    7: (* Wait 2 Seconds After Closing the Last Bin *)
        Active_Material_ID := 0;
        Active_Bin_ID := 0;
        Active_Target_Weight := 0.0;
        Status_Message := 'Settling Delay';
        Completion_Timer(IN := TRUE, PT := Post_Complete_Delay);
        IF Completion_Timer.Q THEN
            Completion_Timer(IN := FALSE);
            Step := 8; // Proceed to reset last weight
        END_IF;
        
    8: (* Reset bin_last_weight to 0 & Complete *)
        Active_Material_ID := 0;
        Active_Bin_ID := 0;
        Active_Target_Weight := 0.0;
        Status_Message := 'Sequence Completed';
        bin_last_weight := 0.0;
        Sequence_Complete := TRUE;
        
        IF NOT Start_Button THEN
            Step := 0;
            Sequence_Complete := FALSE;
            (* Reset all actual weights at completion once start is released *)
            FOR i := 1 TO 6 DO
                Actual_Weights[i] := 0.0;
            END_FOR;
        END_IF;
END_CASE;

END_FUNCTION_BLOCK

// PLC_AC500_V3/Application/old_version/Semi_Auto_Batching_V11
FUNCTION_BLOCK Semi_Auto_Batching_V11
VAR_INPUT
    Start_Button : BOOL;      // Signal to start/resume the batching sequence
    E_Stop_Active : BOOL;     // Emergency Stop (Pause/Hold signal)
    Reset : BOOL;             // Hard reset sequence back to idle state
    Semi_Auto_Bin_Material_Mapping : ARRAY[1..10] OF INT; // Material index mapping for 10 manual silos
    Semi_Auto_Bin_Cutoff_Weights : ARRAY[1..10] OF REAL; // Cutoff weight thresholds (kg)
    Semi_Auto_Bin_Tolerance : ARRAY[1..10] OF REAL; // Tolerance weight offset values (kg)
END_VAR
VAR_IN_OUT
    load_cell_value : REAL;   // Weight value read/written from load cell
END_VAR
VAR_OUTPUT
    Semi_Auto_Bin : ARRAY[1..10] OF BOOL; // Prompts/indicators for Bins 7..16
    semi_auto_bin_cutoff : ARRAY[1..10] OF BOOL; // Manual pre-cutoff indicators
    semi_auto_bin_motor : ARRAY[1..10] OF BOOL; // Main manual feeder motor outputs
    Actual_Weights : ARRAY[1..10] OF REAL; // Actual weight poured per silo
    Sequence_Complete : BOOL;  // Batch complete flag
    Active_Material_ID : INT;  // Currently active ingredient ID
    Active_Bin_ID : INT;       // Currently active physical Bin ID (7..16)
    Active_Target_Weight : REAL; // Recipe target weight of active bin (with tolerance applied)
    Error_Code : INT;          // Active error code
    Status_Message : STRING;   // Diagnostic text message
END_VAR
VAR
    Step : INT := 0;          // State machine index (0: Idle, 1..10: Bins, 11..20: Delays, 30: Settling, 40: Complete)
    bin_last_weight : REAL;   // Baseline weight snapshot before starting current bin
    actual_bin : REAL;        // Current weight added from active bin
    target_act_bin : REAL;    // Effective target weight to add from the active bin (GVL target - Tolerance)
    cutoff_trigger_weight : REAL; // Calculated target threshold weight minus cutoff and tolerance values
    Paused_By_EStop : BOOL := FALSE; // Pause status latch
    
    Mat_Idx : INT;
    i : INT;                  // General loop index
    
    (* TIMERS FOR TRANSITIONS & DELAYS *)
    Transition_Timer : TON;
    Completion_Timer : TON;
    Operator_Timer : TON;
    Step_Delay_Time : TIME := T#2S;
    Post_Complete_Delay : TIME := T#2S;
    
    (* SELF-CONTAINED SIMULATION VARIABLES *)
    Simulation_Mode : BOOL := TRUE;
    Sim_Rate : REAL := 10.0;            // Simulated pouring speed (10.0 kg/s)
    Sim_Timer : TON;
    Start_Sim_Weight : REAL;
    Discharge_Active : BOOL;
END_VAR

(* Semi-Auto Batching FB V11 with E-Stop Pause & Reset Logic *)

(* 1. HARD RESET INTERLOCK (Resets weights immediately) *)
IF Reset THEN
    FOR i := 1 TO 10 DO
        Semi_Auto_Bin[i] := FALSE;
        semi_auto_bin_cutoff[i] := FALSE;
        semi_auto_bin_motor[i] := FALSE;
        Actual_Weights[i] := 0.0;
    END_FOR;
    Sequence_Complete := FALSE;
    Active_Material_ID := 0;
    Active_Bin_ID := 0;
    Active_Target_Weight := 0.0;
    Error_Code := 0;
    Status_Message := 'Semi-Auto Reset Activated';
    Paused_By_EStop := FALSE;
    Step := 0;
    
    (* Clear simulation weights immediately *)
    load_cell_value := 0.0;
    bin_last_weight := 0.0;
    Start_Sim_Weight := 0.0;
    
    Transition_Timer(IN := FALSE);
    Completion_Timer(IN := FALSE);
    Operator_Timer(IN := FALSE);
    Sim_Timer(IN := FALSE);
    RETURN;
END_IF;

(* 2. E-STOP PAUSE / HOLD LOGIC *)
IF E_Stop_Active THEN
    Paused_By_EStop := TRUE;
END_IF;

IF Paused_By_EStop THEN
    (* Suspend all indicators and feeder outputs *)
    FOR i := 1 TO 10 DO
        Semi_Auto_Bin[i] := FALSE;
        semi_auto_bin_cutoff[i] := FALSE;
        semi_auto_bin_motor[i] := FALSE;
    END_FOR;
    
    IF E_Stop_Active THEN
        Status_Message := 'Semi-Auto Paused: Emergency Stop Active!';
    ELSE
        Status_Message := 'Semi-Auto Paused: Press Start to Resume';
        
        (* Resume sequence when Start Button is pressed *)
        IF Start_Button THEN
            Paused_By_EStop := FALSE;
        END_IF;
    END_IF;
    
    (* Freeze simulation and safety timers *)
    Sim_Timer(IN := FALSE);
    Transition_Timer(IN := FALSE);
    Completion_Timer(IN := FALSE);
    Operator_Timer(IN := FALSE);
    RETURN;
END_IF;

(* 3. SELF-CONTAINED SIMULATION WEIGHT MANAGEMENT *)
IF Simulation_Mode THEN
    (* Reset simulation to baseline *)
    IF Step = 0 AND NOT Start_Button AND NOT Sequence_Complete THEN
        load_cell_value := 0.0;
        bin_last_weight := 0.0;
        Start_Sim_Weight := 0.0;
        Sim_Timer(IN := FALSE);
    END_IF;
    
    (* Check if operator is actively pouring *)
    Discharge_Active := FALSE;
    IF Step >= 1 AND Step <= 10 THEN
        Discharge_Active := semi_auto_bin_motor[Step];
    END_IF;
    
    (* Simulate weight gain on the load cell *)
    IF Discharge_Active THEN
        Sim_Timer(IN := TRUE, PT := T#1000S);
        load_cell_value := Start_Sim_Weight + (TIME_TO_REAL(Sim_Timer.ET) / 1000.0) * Sim_Rate;
    ELSE
        Sim_Timer(IN := FALSE);
        Start_Sim_Weight := load_cell_value;
    END_IF;
END_IF;


(* 4. RECIPE SEQUENCE START *)
IF Step = 0 AND Start_Button THEN
    Step := 1;
    bin_last_weight := load_cell_value;
    Sequence_Complete := FALSE;
    Error_Code := 0;
    Status_Message := 'Semi-Auto Pour Started';
    Active_Target_Weight := 0.0;
    (* Clear actual weights on start *)
    FOR i := 1 TO 10 DO
        Actual_Weights[i] := 0.0;
        Semi_Auto_Bin[i] := FALSE;
        semi_auto_bin_cutoff[i] := FALSE;
        semi_auto_bin_motor[i] := FALSE;
    END_FOR;
END_IF;


(* 5. SEQUENCE CONTROL STATE MACHINE *)
CASE Step OF
    0:
        Active_Material_ID := 0;
        Active_Bin_ID := 0;
        Active_Target_Weight := 0.0;
        IF Error_Code = 0 THEN Status_Message := 'Semi-Auto Idle'; END_IF;
        
    1..10: (* Prompts Silos 7 to 16 *)
        Mat_Idx := Semi_Auto_Bin_Material_Mapping[Step];
        
        (* Skip this step instantly if material mapping is 0 OR target weight is 0.0 kg *)
        IF Mat_Idx = 0 OR (Mat_Idx <= 20 AND GVL.Recipe_Weights[Mat_Idx] = 0.0) THEN
            Step := Step + 1;
        ELSE
            (* Calculate effective target weight (Looked up Target - Tolerance) *)
            target_act_bin := GVL.Recipe_Weights[Mat_Idx] - Semi_Auto_Bin_Tolerance[Step];
            Active_Target_Weight := target_act_bin;
            
            (* Calculate weight added by current active bin *)
            actual_bin := load_cell_value - bin_last_weight;
            Actual_Weights[Step] := actual_bin;
            
            (* Calculate cutoff trigger threshold *)
            cutoff_trigger_weight := target_act_bin - Semi_Auto_Bin_Cutoff_Weights[Step];
            
            Active_Material_ID := Mat_Idx;
            Active_Bin_ID := Step;
            Status_Message := 'Semi-Auto Pouring Active';
            
            (* COARSE/FINE FEED TRANSITIONS WITH TOLERANCE OFFSETS *)
            IF actual_bin < cutoff_trigger_weight THEN
                (* Phase 1: Coarse Feed *)
                Semi_Auto_Bin[Step] := TRUE;
                semi_auto_bin_cutoff[Step] := FALSE;
                semi_auto_bin_motor[Step] := TRUE;
            ELSIF actual_bin < target_act_bin THEN
                (* Phase 2: Fine Feed *)
                Semi_Auto_Bin[Step] := FALSE;
                semi_auto_bin_cutoff[Step] := TRUE;
                semi_auto_bin_motor[Step] := TRUE;
            ELSE
                (* Phase 3: Completed (All OFF) *)
                Semi_Auto_Bin[Step] := FALSE;
                semi_auto_bin_cutoff[Step] := FALSE;
                semi_auto_bin_motor[Step] := FALSE;
                bin_last_weight := load_cell_value;
                Active_Target_Weight := 0.0;
                Step := 10 + Step; // Offset to separate transition states
            END_IF;
            
            (* RUNTIME CHECKS *)
            (* Check 21 & 22: Scale Limits *)
            IF load_cell_value > 500.0 THEN
                Error_Code := 21;
                Status_Message := 'Error 21: Scale Overloaded!';
                Paused_By_EStop := TRUE;
            ELSIF load_cell_value < 0.0 THEN
                Error_Code := 22;
                Status_Message := 'Error 22: Scale Underloaded/Fault!';
                Paused_By_EStop := TRUE;
            END_IF;
            
            (* Check 30: Operator Timeout *)
            Operator_Timer(IN := semi_auto_bin_motor[Step], PT := T#300S);
            IF Operator_Timer.Q THEN
                Error_Code := 30;
                Status_Message := 'Error 30: Semi-Auto Operator Timeout!';
                Paused_By_EStop := TRUE;
            END_IF;
        END_IF;

    11..19: (* Transition Delays (Between Bins) *)
        Active_Material_ID := 0;
        Active_Bin_ID := 0;
        Active_Target_Weight := 0.0;
        Status_Message := 'Transition Delay';
        Transition_Timer(IN := TRUE, PT := Step_Delay_Time);
        IF Transition_Timer.Q THEN
            Transition_Timer(IN := FALSE);
            Step := (Step - 10) + 1; // Advance to next bin
        END_IF;
        
    20: (* Transition Delay After Last Bin (Bin 10) Closes *)
        Active_Material_ID := 0;
        Active_Bin_ID := 0;
        Active_Target_Weight := 0.0;
        Status_Message := 'Settling Last Bin';
        Transition_Timer(IN := TRUE, PT := Step_Delay_Time);
        IF Transition_Timer.Q THEN
            Transition_Timer(IN := FALSE);
            Step := 30; // Go to post-discharge wait step (State 30)
        END_IF;

    30: (* Wait 2 Seconds After Closing the Last Bin *)
        Active_Material_ID := 0;
        Active_Bin_ID := 0;
        Active_Target_Weight := 0.0;
        Status_Message := 'Settling Delay';
        Completion_Timer(IN := TRUE, PT := Post_Complete_Delay);
        IF Completion_Timer.Q THEN
            Completion_Timer(IN := FALSE);
            Step := 40; // Proceed to reset last weight (State 40)
        END_IF;
        
    40: (* Reset bin_last_weight to 0 & Complete *)
        Active_Material_ID := 0;
        Active_Bin_ID := 0;
        Active_Target_Weight := 0.0;
        Status_Message := 'Sequence Completed';
        bin_last_weight := 0.0;
        Sequence_Complete := TRUE;
        
        IF NOT Start_Button THEN
            Step := 0;
            Sequence_Complete := FALSE;
            (* Reset all actual weights at completion once start is released *)
            FOR i := 1 TO 10 DO
                Actual_Weights[i] := 0.0;
            END_FOR;
        END_IF;
END_CASE;

END_FUNCTION_BLOCK

// PLC_AC500_V3/Application/old_version/Auto_Batching_V12
FUNCTION_BLOCK Auto_Batching_V12
VAR_INPUT
    Start_Button : BOOL;      // Signal to start/resume the batching sequence
    E_Stop_Active : BOOL;     // Emergency Stop (Pause/Hold signal)
    Reset : BOOL;             // Hard reset sequence back to idle state
    Auto_Bin_Material_Mapping : ARRAY[1..6] OF INT; // Material index mapping for 6 bins
    Auto_Bin_Cutoff_Weights : ARRAY[1..6] OF REAL; // Cutoff weight thresholds (kg)
    Auto_Bin_Tolerance : ARRAY[1..6] OF REAL; // Tolerance weight offset values (kg)
END_VAR
VAR_IN_OUT
    load_cell_value : REAL;   // Weight value read/written from load cell
END_VAR
VAR_OUTPUT
    Auto_Bin : ARRAY[1..6] OF BOOL; // Coarse feed valve outputs
    auto_bin_cutoff : ARRAY[1..6] OF BOOL; // Fine feed cutoff trigger indicators
    auto_bin_motor : ARRAY[1..6] OF BOOL; // Main conveyor motor outputs
    Actual_Weights : ARRAY[1..6] OF REAL; // Actual weight poured per silo
    Sequence_Complete : BOOL;  // Batch complete flag
    Active_Material_ID : INT;  // Currently active ingredient ID
    Active_Bin_ID : INT;       // Currently active physical Bin ID (1..6)
    Active_Target_Weight : REAL; // Recipe target weight of active bin (with tolerance applied)
    Error_Code : INT;          // Active error code
    Status_Message : STRING;   // Diagnostic text message
END_VAR
VAR
    Step : INT;                // State machine index
    bin_last_weight : REAL;   // Baseline weight snapshot before starting current bin
    actual_bin : REAL;        // Current weight added from active bin
    target_act_bin : REAL;    // Effective target weight to add from the active bin
    cutoff_trigger_weight : REAL; // Calculated trigger weight
    Paused_By_EStop : BOOL;    // Pause status latch
    
    Mat_Idx : INT;
    i : INT;                  // General loop index
    
    (* TIMERS FOR TRANSITIONS & DELAYS *)
    Transition_Timer : TON;
    Completion_Timer : TON;
    
    (* SELF-CONTAINED SIMULATION VARIABLES *)
    Simulation_Mode : BOOL;    // Simulation disabled
    Sim_Rate : REAL;
    Sim_Timer : TON;
    Start_Sim_Weight : REAL;
    Discharge_Active : BOOL;
END_VAR

(* Auto Batching FB V12 with E-Stop Pause & Reset Logic *)

(* 1. HARD RESET INTERLOCK (Resets weights immediately) *)
IF Reset THEN
    FOR i := 1 TO 6 DO
        Auto_Bin[i] := FALSE;
        auto_bin_cutoff[i] := FALSE;
        auto_bin_motor[i] := FALSE;
        Actual_Weights[i] := 0.0;
    END_FOR;
    Sequence_Complete := FALSE;
    Active_Material_ID := 0;
    Active_Bin_ID := 0;
    Active_Target_Weight := 0.0;
    Error_Code := 0;
    Status_Message := '';
    Paused_By_EStop := FALSE;
    Step := 0;
    
    load_cell_value := 0.0;
    bin_last_weight := 0.0;
    Start_Sim_Weight := 0.0;
    
    Transition_Timer(IN := FALSE);
    Completion_Timer(IN := FALSE);
    Sim_Timer(IN := FALSE);
    RETURN;
END_IF;

(* 2. E-STOP PAUSE / HOLD LOGIC *)
IF E_Stop_Active THEN
    Paused_By_EStop := TRUE;
END_IF;

IF Paused_By_EStop THEN
    (* Suspend all valve/motor control outputs immediately *)
    FOR i := 1 TO 6 DO
        Auto_Bin[i] := FALSE;
        auto_bin_cutoff[i] := FALSE;
        auto_bin_motor[i] := FALSE;
    END_FOR;
    
    IF E_Stop_Active THEN
        Status_Message := 'Auto Paused: Emergency Stop Active!';
    ELSE
        Status_Message := 'Auto Paused: Press Start to Resume';
        
        (* Resume sequence when Start Button is pressed *)
        IF Start_Button THEN
            Paused_By_EStop := FALSE;
        END_IF;
    END_IF;
    
    (* Freeze simulation timers and exit code execution *)
    Sim_Timer(IN := FALSE);
    Transition_Timer(IN := FALSE);
    Completion_Timer(IN := FALSE);
    RETURN;
END_IF;

(* 3. SELF-CONTAINED SIMULATION WEIGHT MANAGEMENT *)
IF Simulation_Mode THEN
    (* Reset simulation to baseline *)
    IF Step = 0 AND NOT Start_Button AND NOT Sequence_Complete THEN
        load_cell_value := 0.0;
        bin_last_weight := 0.0;
        Start_Sim_Weight := 0.0;
        Sim_Timer(IN := FALSE);
    END_IF;
    
    (* Check if any valve is actively discharging *)
    Discharge_Active := FALSE;
    IF Step >= 1 AND Step <= 6 THEN
        Discharge_Active := auto_bin_motor[Step];
    END_IF;
    
    (* Simulate weight gain on the load cell *)
    IF Discharge_Active THEN
        Sim_Timer(IN := TRUE, PT := T#1000S);
        load_cell_value := Start_Sim_Weight + (TIME_TO_REAL(Sim_Timer.ET) / 1000.0) * Sim_Rate;
    ELSE
        Sim_Timer(IN := FALSE);
        Start_Sim_Weight := load_cell_value;
    END_IF;
END_IF;


(* 4. RECIPE SEQUENCE START *)
IF Step = 0 AND Start_Button THEN
    Step := 1;
    bin_last_weight := load_cell_value;
    Sequence_Complete := FALSE;
    Error_Code := 0;
    Status_Message := 'Auto Pour Started';
    Active_Target_Weight := 0.0;
    (* Clear actual weights and outputs on start *)
    FOR i := 1 TO 6 DO
        Actual_Weights[i] := 0.0;
        Auto_Bin[i] := FALSE;
        auto_bin_cutoff[i] := FALSE;
        auto_bin_motor[i] := FALSE;
    END_FOR;
END_IF;


(* 5. SEQUENCE CONTROL STATE MACHINE *)
CASE Step OF
    0:
        Active_Material_ID := 0;
        Active_Bin_ID := 0;
        Active_Target_Weight := 0.0;
        IF Error_Code = 0 THEN Status_Message := 'Auto Idle'; END_IF;
        
    1..6: (* Discharging Silos 1 to 6 *)
        Mat_Idx := Auto_Bin_Material_Mapping[Step];
        
        (* Skip this step instantly if material mapping is 0 OR target weight is 0.0 kg *)
        IF Mat_Idx = 0 OR (Mat_Idx <= 20 AND GVL.Recipe_Weights[Mat_Idx] = 0.0) THEN
            Step := Step + 1;
        ELSE
            (* Calculate effective target weight (Looked up Target - Tolerance) *)
            target_act_bin := GVL.Recipe_Weights[Mat_Idx] - Auto_Bin_Tolerance[Step];
            Active_Target_Weight := target_act_bin;
            
            (* Calculate weight added by current active bin *)
            actual_bin := load_cell_value - bin_last_weight;
            Actual_Weights[Step] := actual_bin;
            
            (* Calculate cutoff trigger threshold *)
            cutoff_trigger_weight := target_act_bin - Auto_Bin_Cutoff_Weights[Step];
            
            Active_Material_ID := Mat_Idx;
            Active_Bin_ID := Step;
            Status_Message := 'Auto Pouring';
            
            (* COARSE/FINE FEED TRANSITIONS WITH TOLERANCE OFFSETS *)
            IF actual_bin < cutoff_trigger_weight THEN
                (* Phase 1: Coarse Feed *)
                Auto_Bin[Step] := TRUE;
                auto_bin_cutoff[Step] := FALSE;
                auto_bin_motor[Step] := TRUE;
            ELSIF actual_bin < target_act_bin THEN
                (* Phase 2: Fine Feed *)
                Auto_Bin[Step] := FALSE;
                auto_bin_cutoff[Step] := TRUE;
                auto_bin_motor[Step] := TRUE;
            ELSE
                (* Phase 3: Completed (All OFF) *)
                Auto_Bin[Step] := FALSE;
                auto_bin_cutoff[Step] := FALSE;
                auto_bin_motor[Step] := FALSE;
                bin_last_weight := load_cell_value;
                Active_Target_Weight := 0.0;
                Step := 10 + Step; // Offset to separate transition states
            END_IF;
            
            (* RUNTIME CHECKS *)
            (* Check 21 & 22: Scale Limits *)
            IF load_cell_value > 500.0 THEN
                Error_Code := 21;
                Status_Message := 'Error 21: Scale Overloaded!';
                Sequence_Complete := TRUE; // Mark complete on halt
                Paused_By_EStop := TRUE; // Pause sequence on fault
            ELSIF load_cell_value < 0.0 THEN
                Error_Code := 22;
                Status_Message := 'Error 22: Scale Underloaded/Fault!';
                Sequence_Complete := TRUE; // Mark complete on halt
                Paused_By_EStop := TRUE; // Pause sequence on fault
            END_IF;
        END_IF;

    11..15: (* Transition Delays (Between Bins) *)
        Active_Material_ID := 0;
        Active_Bin_ID := 0;
        Active_Target_Weight := 0.0;
        Status_Message := 'Transition Delay';
        
        Transition_Timer(IN := TRUE, PT := T#2S);
        IF Transition_Timer.Q THEN
            Transition_Timer(IN := FALSE);
            Step := (Step - 10) + 1; // Advance to next bin
        END_IF;
        
    16: (* Transition Delay After Last Bin (Bin 6) Closes *)
        Active_Material_ID := 0;
        Active_Bin_ID := 0;
        Active_Target_Weight := 0.0;
        Status_Message := 'Settling Last Bin';
        
        Transition_Timer(IN := TRUE, PT := T#2S);
        IF Transition_Timer.Q THEN
            Transition_Timer(IN := FALSE);
            Step := 7; // Go to post-discharge wait step
        END_IF;

    7: (* Wait 2 Seconds After Closing the Last Bin *)
        Active_Material_ID := 0;
        Active_Bin_ID := 0;
        Active_Target_Weight := 0.0;
        Status_Message := 'Settling Delay';
        Completion_Timer(IN := TRUE, PT := T#2S);
        IF Completion_Timer.Q THEN
            Completion_Timer(IN := FALSE);
            Step := 8; // Proceed to reset last weight
        END_IF;
        
    8: (* Reset bin_last_weight to 0 & Complete *)
        Active_Material_ID := 0;
        Active_Bin_ID := 0;
        Active_Target_Weight := 0.0;
        Status_Message := 'Sequence Completed';
        bin_last_weight := 0.0;
        Sequence_Complete := TRUE;
        
        IF NOT Start_Button THEN
            Step := 0;
            Sequence_Complete := FALSE;
            (* Reset all actual weights at completion once start is released *)
            FOR i := 1 TO 6 DO
                Actual_Weights[i] := 0.0;
            END_FOR;
        END_IF;
END_CASE;

END_FUNCTION_BLOCK

// PLC_AC500_V3/Application/old_version/Semi_Auto_Batching_V12
FUNCTION_BLOCK Semi_Auto_Batching_V12
VAR_INPUT
    Start_Button : BOOL;      // Signal to start/resume the batching sequence
    E_Stop_Active : BOOL;     // Emergency Stop (Pause/Hold signal)
    Reset : BOOL;             // Hard reset sequence back to idle state
    Semi_Auto_Bin_Material_Mapping : ARRAY[1..10] OF INT; // Material index mapping for 10 manual silos
    Semi_Auto_Bin_Cutoff_Weights : ARRAY[1..10] OF REAL; // Cutoff weight thresholds (kg)
    Semi_Auto_Bin_Tolerance : ARRAY[1..10] OF REAL; // Tolerance weight offset values (kg)
END_VAR
VAR_IN_OUT
    load_cell_value : REAL;   // Weight value read/written from load cell
END_VAR
VAR_OUTPUT
    Semi_Auto_Bin : ARRAY[1..10] OF BOOL; // Prompts/indicators for Bins 7..16
    semi_auto_bin_cutoff : ARRAY[1..10] OF BOOL; // Manual pre-cutoff indicators
    semi_auto_bin_motor : ARRAY[1..10] OF BOOL; // Main manual feeder motor outputs
    Actual_Weights : ARRAY[1..10] OF REAL; // Actual weight poured per silo
    Sequence_Complete : BOOL;  // Batch complete flag
    Active_Material_ID : INT;  // Currently active ingredient ID
    Active_Bin_ID : INT;       // Currently active physical Bin ID (7..16)
    Active_Target_Weight : REAL; // Recipe target weight of active bin (with tolerance applied)
    Error_Code : INT;          // Active error code
    Status_Message : STRING;   // Diagnostic text message
END_VAR
VAR
    Step : INT;                // State machine index
    bin_last_weight : REAL;   // Baseline weight snapshot before starting current bin
    actual_bin : REAL;        // Current weight added from active bin
    target_act_bin : REAL;    // Effective target weight to add from the active bin
    cutoff_trigger_weight : REAL; // Calculated target threshold weight
    Paused_By_EStop : BOOL;    // Pause status latch
    
    Mat_Idx : INT;
    i : INT;                  // General loop index
    
    (* TIMERS FOR TRANSITIONS & DELAYS *)
    Transition_Timer : TON;
    Completion_Timer : TON;
    Operator_Timer : TON;
    
    (* SELF-CONTAINED SIMULATION VARIABLES *)
    Simulation_Mode : BOOL;    // Simulation disabled
    Sim_Rate : REAL;
    Sim_Timer : TON;
    Start_Sim_Weight : REAL;
    Discharge_Active : BOOL;
END_VAR

(* Semi-Auto Batching FB V12 with E-Stop Pause & Reset Logic *)

(* 1. HARD RESET INTERLOCK (Resets weights immediately) *)
IF Reset THEN
    FOR i := 1 TO 10 DO
        Semi_Auto_Bin[i] := FALSE;
        semi_auto_bin_cutoff[i] := FALSE;
        semi_auto_bin_motor[i] := FALSE;
        Actual_Weights[i] := 0.0;
    END_FOR;
    Sequence_Complete := FALSE;
    Active_Material_ID := 0;
    Active_Bin_ID := 0;
    Active_Target_Weight := 0.0;
    Error_Code := 0;
    Status_Message := '';
    Paused_By_EStop := FALSE;
    Step := 0;
    
    load_cell_value := 0.0;
    bin_last_weight := 0.0;
    Start_Sim_Weight := 0.0;
    
    Transition_Timer(IN := FALSE);
    Completion_Timer(IN := FALSE);
    Operator_Timer(IN := FALSE);
    Sim_Timer(IN := FALSE);
    RETURN;
END_IF;

(* 2. E-STOP PAUSE / HOLD LOGIC *)
IF E_Stop_Active THEN
    Paused_By_EStop := TRUE;
END_IF;

IF Paused_By_EStop THEN
    (* Suspend all indicators and feeder outputs *)
    FOR i := 1 TO 10 DO
        Semi_Auto_Bin[i] := FALSE;
        semi_auto_bin_cutoff[i] := FALSE;
        semi_auto_bin_motor[i] := FALSE;
    END_FOR;
    
    IF E_Stop_Active THEN
        Status_Message := 'Semi-Auto Paused: Emergency Stop Active!';
    ELSE
        Status_Message := 'Semi-Auto Paused: Press Start to Resume';
        
        (* Resume sequence when Start Button is pressed *)
        IF Start_Button THEN
            Paused_By_EStop := FALSE;
        END_IF;
    END_IF;
    
    (* Freeze simulation and safety timers *)
    Sim_Timer(IN := FALSE);
    Transition_Timer(IN := FALSE);
    Completion_Timer(IN := FALSE);
    Operator_Timer(IN := FALSE);
    RETURN;
END_IF;

(* 3. SELF-CONTAINED SIMULATION WEIGHT MANAGEMENT *)
IF Simulation_Mode THEN
    (* Reset simulation to baseline *)
    IF Step = 0 AND NOT Start_Button AND NOT Sequence_Complete THEN
        load_cell_value := 0.0;
        bin_last_weight := 0.0;
        Start_Sim_Weight := 0.0;
        Sim_Timer(IN := FALSE);
    END_IF;
    
    (* Check if operator is actively pouring *)
    Discharge_Active := FALSE;
    IF Step >= 1 AND Step <= 10 THEN
        Discharge_Active := semi_auto_bin_motor[Step];
    END_IF;
    
    (* Simulate weight gain on the load cell *)
    IF Discharge_Active THEN
        Sim_Timer(IN := TRUE, PT := T#1000S);
        load_cell_value := Start_Sim_Weight + (TIME_TO_REAL(Sim_Timer.ET) / 1000.0) * Sim_Rate;
    ELSE
        Sim_Timer(IN := FALSE);
        Start_Sim_Weight := load_cell_value;
    END_IF;
END_IF;


(* 4. RECIPE SEQUENCE START *)
IF Step = 0 AND Start_Button THEN
    Step := 1;
    bin_last_weight := load_cell_value;
    Sequence_Complete := FALSE;
    Error_Code := 0;
    Status_Message := 'Semi-Auto Pour Started';
    Active_Target_Weight := 0.0;
    (* Clear actual weights on start *)
    FOR i := 1 TO 10 DO
        Actual_Weights[i] := 0.0;
        Semi_Auto_Bin[i] := FALSE;
        semi_auto_bin_cutoff[i] := FALSE;
        semi_auto_bin_motor[i] := FALSE;
    END_FOR;
END_IF;


(* 5. SEQUENCE CONTROL STATE MACHINE *)
CASE Step OF
    0:
        Active_Material_ID := 0;
        Active_Bin_ID := 0;
        Active_Target_Weight := 0.0;
        IF Error_Code = 0 THEN Status_Message := 'Semi-Auto Idle'; END_IF;
        
    1..10: (* Prompts Silos 7 to 16 *)
        Mat_Idx := Semi_Auto_Bin_Material_Mapping[Step];
        
        (* Skip this step instantly if material mapping is 0 OR target weight is 0.0 kg *)
        IF Mat_Idx = 0 OR (Mat_Idx <= 20 AND GVL.Recipe_Weights[Mat_Idx] = 0.0) THEN
            Step := Step + 1;
        ELSE
            (* Calculate effective target weight (Looked up Target - Tolerance) *)
            target_act_bin := GVL.Recipe_Weights[Mat_Idx] - Semi_Auto_Bin_Tolerance[Step];
            Active_Target_Weight := target_act_bin;
            
            (* Calculate weight added by current active bin *)
            actual_bin := load_cell_value - bin_last_weight;
            Actual_Weights[Step] := actual_bin;
            
            (* Calculate cutoff trigger threshold *)
            cutoff_trigger_weight := target_act_bin - Semi_Auto_Bin_Cutoff_Weights[Step];
            
            Active_Material_ID := Mat_Idx;
            Active_Bin_ID := Step;
            Status_Message := 'Semi-Auto Pouring Active';
            
            (* COARSE/FINE FEED TRANSITIONS WITH TOLERANCE OFFSETS *)
            IF actual_bin < cutoff_trigger_weight THEN
                (* Phase 1: Coarse Feed *)
                Semi_Auto_Bin[Step] := TRUE;
                semi_auto_bin_cutoff[Step] := FALSE;
                semi_auto_bin_motor[Step] := TRUE;
            ELSIF actual_bin < target_act_bin THEN
                (* Phase 2: Fine Feed *)
                Semi_Auto_Bin[Step] := FALSE;
                semi_auto_bin_cutoff[Step] := TRUE;
                semi_auto_bin_motor[Step] := TRUE;
            ELSE
                (* Phase 3: Completed (All OFF) *)
                Semi_Auto_Bin[Step] := FALSE;
                semi_auto_bin_cutoff[Step] := FALSE;
                semi_auto_bin_motor[Step] := FALSE;
                bin_last_weight := load_cell_value;
                Active_Target_Weight := 0.0;
                Step := 10 + Step; // Offset to separate transition states
            END_IF;
            
            (* RUNTIME CHECKS *)
            (* Check 21 & 22: Scale Limits *)
            IF load_cell_value > 500.0 THEN
                Error_Code := 21;
                Status_Message := 'Error 21: Scale Overloaded!';
                Sequence_Complete := TRUE; // Mark complete on halt
                Paused_By_EStop := TRUE;
            ELSIF load_cell_value < 0.0 THEN
                Error_Code := 22;
                Status_Message := 'Error 22: Scale Underloaded/Fault!';
                Sequence_Complete := TRUE; // Mark complete on halt
                Paused_By_EStop := TRUE;
            END_IF;
            
            (* Check 30: Operator Timeout *)
            Operator_Timer(IN := semi_auto_bin_motor[Step], PT := T#300S);
            IF Operator_Timer.Q THEN
                Error_Code := 30;
                Status_Message := 'Error 30: Semi-Auto Operator Timeout!';
                Sequence_Complete := TRUE; // Mark complete on halt
                Paused_By_EStop := TRUE;
            END_IF;
        END_IF;

    11..19: (* Transition Delays (Between Bins) *)
        Active_Material_ID := 0;
        Active_Bin_ID := 0;
        Active_Target_Weight := 0.0;
        Status_Message := 'Transition Delay';
        Transition_Timer(IN := TRUE, PT := T#2S);
        IF Transition_Timer.Q THEN
            Transition_Timer(IN := FALSE);
            Step := (Step - 10) + 1; // Advance to next bin
        END_IF;
        
    20: (* Transition Delay After Last Bin (Bin 10) Closes *)
        Active_Material_ID := 0;
        Active_Bin_ID := 0;
        Active_Target_Weight := 0.0;
        Status_Message := 'Settling Last Bin';
        Transition_Timer(IN := TRUE, PT := T#2S);
        IF Transition_Timer.Q THEN
            Transition_Timer(IN := FALSE);
            Step := 30; // Go to post-discharge wait step (State 30)
        END_IF;

    30: (* Wait 2 Seconds After Closing the Last Bin *)
        Active_Material_ID := 0;
        Active_Bin_ID := 0;
        Active_Target_Weight := 0.0;
        Status_Message := 'Settling Delay';
        Completion_Timer(IN := TRUE, PT := T#2S);
        IF Completion_Timer.Q THEN
            Completion_Timer(IN := FALSE);
            Step := 40; // Proceed to reset last weight (State 40)
        END_IF;
        
    40: (* Reset bin_last_weight to 0 & Complete *)
        Active_Material_ID := 0;
        Active_Bin_ID := 0;
        Active_Target_Weight := 0.0;
        Status_Message := 'Sequence Completed';
        bin_last_weight := 0.0;
        Sequence_Complete := TRUE;
        
        IF NOT Start_Button THEN
            Step := 0;
            Sequence_Complete := FALSE;
            (* Reset all actual weights at completion once start is released *)
            FOR i := 1 TO 10 DO
                Actual_Weights[i] := 0.0;
            END_FOR;
        END_IF;
END_CASE;

END_FUNCTION_BLOCK

// PLC_AC500_V3/Application/old_version/batching12
PROGRAM batching12
VAR
    Auto_Ctrl : Auto_Batching_V12;
    Semi_Auto_Ctrl : Semi_Auto_Batching_V12;
    
    (* Sub-Block Diagnostic Indicators (not in GVL) *)
    Auto_Active_Target : REAL; // Active Target Weight for Auto (displays GVL setpoint - Tolerance)
    Auto_Err : INT;
    Auto_Msg : STRING;
    
    Semi_Auto_Active_Target : REAL; // Active Target Weight for Semi-Auto (displays GVL setpoint - Tolerance)
    Semi_Auto_Err : INT;
    Semi_Auto_Msg : STRING;
    
    (* Process Outputs *)
    Auto_Bin : ARRAY[1..6] OF BOOL; // Valve control outputs (Coarse)
    auto_bin_cutoff : ARRAY[1..6] OF BOOL; // Cutoff indicators (Fine)
    auto_bin_motor : ARRAY[1..6] OF BOOL; // Conveyor/feeder motor outputs
    
    Semi_Auto_Bin : ARRAY[1..10] OF BOOL; // Prompt indicators (Coarse)
    semi_auto_bin_cutoff : ARRAY[1..10] OF BOOL; // Cutoff indicators (Fine)
    semi_auto_bin_motor : ARRAY[1..10] OF BOOL; // Conveyor/feeder motor outputs
    
    Auto_Weights : ARRAY[1..6] OF REAL;
    Semi_Auto_Weights : ARRAY[1..10] OF REAL;
    
    Auto_Complete : BOOL;
    Semi_Auto_Complete : BOOL;
    
    (* Repetitive Cycle Status (not in GVL) *)
    Completed_Batch_Cycles : INT;      // Total completed batch cycle loops
    All_Cycles_Complete : BOOL;         // Indicator for full set completion
    
    (* Diagnostics & Interlocks (not in GVL) *)
    Status_Message : STRING;
    
    i : INT;
    j : INT;
    Duplicate_Found : BOOL;
    Invalid_Material_Range : BOOL;
    Weight_Limit_Error : BOOL;
    
    (* Cycle Manager state variables *)
    Cycle_Manager_State : INT;         // State index for loop management
    Internal_FB_Start : BOOL;          // Controlled command to restart sub-blocks
END_VAR

(* 1. STARTUP CONFIGURATION AND WEIGHT CHECKS *)
Duplicate_Found := FALSE;
Invalid_Material_Range := FALSE;
Weight_Limit_Error := FALSE;

FOR i := 1 TO 6 DO
    (* Check 2: Out of Range (Auto) *)
    IF GVL.Auto_Bin_Material_Mapping[i] < 0 OR GVL.Auto_Bin_Material_Mapping[i] > 20 THEN
        Invalid_Material_Range := TRUE;
    END_IF;
    
    (* Check 1: Duplicate Cross-Array Material ID *)
    IF GVL.Auto_Bin_Material_Mapping[i] <> 0 AND GVL.Auto_Bin_Material_Mapping[i] <= 20 THEN
        FOR j := 1 TO 10 DO
            IF GVL.Auto_Bin_Material_Mapping[i] = GVL.Semi_Auto_Bin_Material_Mapping[j] THEN
                Duplicate_Found := TRUE;
            END_IF;
        END_FOR;
    END_IF;
    
    (* Check 3: Recipe weight is less than Cutoff + Tolerance *)
    IF GVL.Auto_Bin_Material_Mapping[i] <> 0 AND GVL.Auto_Bin_Material_Mapping[i] <= 20 THEN
        IF GVL.Recipe_Weights[GVL.Auto_Bin_Material_Mapping[i]] > 0.0 THEN
            IF GVL.Recipe_Weights[GVL.Auto_Bin_Material_Mapping[i]] < (GVL.Auto_Bin_Cutoff_Weights[i] + GVL.Auto_Bin_Tolerance[i]) THEN
                Weight_Limit_Error := TRUE;
            END_IF;
        END_IF;
    END_IF;
END_FOR;

FOR j := 1 TO 10 DO
    (* Check 2: Out of Range (Semi-Auto) *)
    IF GVL.Semi_Auto_Bin_Material_Mapping[j] < 0 OR GVL.Semi_Auto_Bin_Material_Mapping[j] > 20 THEN
        Invalid_Material_Range := TRUE;
    END_IF;
    
    (* Check 3: Recipe weight check (Semi-Auto) *)
    IF GVL.Semi_Auto_Bin_Material_Mapping[j] <> 0 AND GVL.Semi_Auto_Bin_Material_Mapping[j] <= 20 THEN
        IF GVL.Recipe_Weights[GVL.Semi_Auto_Bin_Material_Mapping[j]] > 0.0 THEN
            IF GVL.Recipe_Weights[GVL.Semi_Auto_Bin_Material_Mapping[j]] < (GVL.Semi_Auto_Bin_Cutoff_Weights[j] + GVL.Semi_Auto_Bin_Tolerance[j]) THEN
                Weight_Limit_Error := TRUE;
            END_IF;
        END_IF;
    END_IF;
END_FOR;

(* Configuration Error Resolution *)
IF Duplicate_Found THEN
    GVL.Error_Code := 1;
    Status_Message := 'Error 1: Duplicate Material ID mapped in Auto and Semi-Auto!';
ELSIF Invalid_Material_Range THEN
    GVL.Error_Code := 2;
    Status_Message := 'Error 2: Material Index configuration out of range (1..20)!';
ELSIF Weight_Limit_Error THEN
    GVL.Error_Code := 3;
    Status_Message := 'Error 3: Recipe weight is less than Cutoff + Tolerance!';
ELSE
    IF GVL.Error_Code <= 3 THEN
        GVL.Error_Code := 0;
    END_IF;
END_IF;

(* Abort/Clear arrays if Configuration error is active or Hard Reset is pressed *)
IF (GVL.Error_Code >= 1 AND GVL.Error_Code <= 3) OR GVL.Reset THEN
    FOR i := 1 TO 6 DO 
        Auto_Bin[i] := FALSE; 
        auto_bin_cutoff[i] := FALSE; 
        auto_bin_motor[i] := FALSE; 
        Auto_Weights[i] := 0.0;
    END_FOR;
    
    FOR i := 1 TO 10 DO 
        Semi_Auto_Bin[i] := FALSE; 
        semi_auto_bin_cutoff[i] := FALSE; 
        semi_auto_bin_motor[i] := FALSE; 
        Semi_Auto_Weights[i] := 0.0;
    END_FOR;
    
    Internal_FB_Start := FALSE;
    Auto_Ctrl(Start_Button := FALSE, E_Stop_Active := FALSE, Reset := GVL.Reset, load_cell_value := GVL.load_cell_auto);
    Semi_Auto_Ctrl(Start_Button := FALSE, E_Stop_Active := FALSE, Reset := GVL.Reset, load_cell_value := GVL.load_cell_semi_auto);
    
    Auto_Active_Target := 0.0;
    Semi_Auto_Active_Target := 0.0;
    
    Auto_Complete := TRUE;
    Semi_Auto_Complete := TRUE;
    All_Cycles_Complete := TRUE;
    
    GVL.Cycle_Hold_Active := FALSE;
    GVL.Run := FALSE;
    Cycle_Manager_State := 0;
    
    IF GVL.Reset THEN
        GVL.Error_Code := 0;
        GVL.Current_Batch_Cycle := 0;
        Completed_Batch_Cycles := 0;
        Status_Message := 'System Reset Activated';
        Auto_Complete := FALSE;
        Semi_Auto_Complete := FALSE;
        All_Cycles_Complete := FALSE;
        
        GVL.Auto_Active_Mat := 0;
        GVL.Auto_Active_Bin := 0;
        GVL.Semi_Auto_Active_Mat := 0;
        GVL.Semi_Auto_Active_Bin := 0;
    END_IF;
    RETURN;
END_IF;


(* 2. REPETITIVE CYCLE MANAGER STATE MACHINE WITH HOLD RELEASE *)
CASE Cycle_Manager_State OF
    0: (* IDLE STATE *)
        Internal_FB_Start := FALSE;
        All_Cycles_Complete := FALSE;
        GVL.Cycle_Hold_Active := FALSE;
        GVL.Run := FALSE;
        IF GVL.Error_Code = 0 THEN Status_Message := 'System Ready'; END_IF;
        
        IF GVL.Start_Button THEN
            GVL.Current_Batch_Cycle := 1;
            Completed_Batch_Cycles := 0;
            
            (* Explicitly reset latch flags so FBs can run fresh *)
            Auto_Complete := FALSE;
            Semi_Auto_Complete := FALSE;
            
            GVL.Run := TRUE;
            Cycle_Manager_State := 1;
        END_IF;
        
    1: (* RUN STATE (Run Sub-Blocks) *)
        Internal_FB_Start := TRUE;
        GVL.Run := TRUE;
        Status_Message := CONCAT('Running Batch Cycle ', INT_TO_STRING(GVL.Current_Batch_Cycle));
        
        (* Monitor completion of active step *)
        IF Auto_Complete AND Semi_Auto_Complete THEN
            Cycle_Manager_State := 2;
        END_IF;
        
    2: (* CHECK REPEAT CYCLE STATE *)
        Completed_Batch_Cycles := GVL.Current_Batch_Cycle;
        GVL.Run := TRUE;
        
        (* Block cycle repeat in case of active error *)
        IF GVL.Current_Batch_Cycle < GVL.Target_Batch_Cycles AND GVL.Error_Code = 0 THEN
            (* Hold cycle loop progression *)
            GVL.Cycle_Hold_Active := TRUE;
            Cycle_Manager_State := 5; // Go to hold wait state
        else
            (* All loop cycles complete *)
            Cycle_Manager_State := 4;
        END_IF;
        
    5: (* PAUSED BETWEEN CYCLES *)
        Internal_FB_Start := TRUE; // Keep FBs active in finished step state
        GVL.Run := TRUE;
        Status_Message := CONCAT('Cycle ', CONCAT(INT_TO_STRING(GVL.Current_Batch_Cycle), ' Complete. Waiting to Release.'));
        
        (* Operator toggles hold status back to FALSE to proceed *)
        IF NOT GVL.Cycle_Hold_Active THEN
            Cycle_Manager_State := 3; // Go to auto-reset pulse
        END_IF;
        
    3: (* AUTO-RESET PULSE (Pulse Start command low to reset state machines) *)
        Internal_FB_Start := FALSE;
        GVL.Run := TRUE;
        Status_Message := 'Resetting Sequence for Next Cycle';
        
        (* Verify sub-blocks have fully reset to idle step *)
        IF NOT Auto_Complete AND NOT Semi_Auto_Complete THEN
            GVL.Current_Batch_Cycle := GVL.Current_Batch_Cycle + 1;
            Cycle_Manager_State := 1; // Start next cycle
        END_IF;
        
    4: (* SEQUENCE FULLY COMPLETED STATE *)
        Internal_FB_Start := FALSE;
        All_Cycles_Complete := TRUE;
        GVL.Run := FALSE;
        Status_Message := 'All Batch Cycles Completed';
        
        IF NOT GVL.Start_Button THEN
            Cycle_Manager_State := 0;
        END_IF;
END_CASE;


(* 3. CONCURRENT EXECUTION OF FB INSTANCES *)
Auto_Ctrl(
    Start_Button := Internal_FB_Start,
    E_Stop_Active := GVL.E_Stop_Active,
    Reset := GVL.Reset,
    load_cell_value := GVL.load_cell_auto,
    Auto_Bin_Material_Mapping := GVL.Auto_Bin_Material_Mapping,
    Auto_Bin_Cutoff_Weights := GVL.Auto_Bin_Cutoff_Weights,
    Auto_Bin_Tolerance := GVL.Auto_Bin_Tolerance,
    Auto_Bin => Auto_Bin,
    auto_bin_cutoff => auto_bin_cutoff,
    auto_bin_motor => auto_bin_motor,
    Actual_Weights => Auto_Weights,
    Sequence_Complete => Auto_Complete,
    Active_Material_ID => GVL.Auto_Active_Mat,
    Active_Bin_ID => GVL.Auto_Active_Bin,
    Active_Target_Weight => Auto_Active_Target,
    Error_Code => Auto_Err,
    Status_Message => Auto_Msg
);

Semi_Auto_Ctrl(
    Start_Button := Internal_FB_Start,
    E_Stop_Active := GVL.E_Stop_Active,
    Reset := GVL.Reset,
    load_cell_value := GVL.load_cell_semi_auto,
    Semi_Auto_Bin_Material_Mapping := GVL.Semi_Auto_Bin_Material_Mapping,
    Semi_Auto_Bin_Cutoff_Weights := GVL.Semi_Auto_Bin_Cutoff_Weights,
    Semi_Auto_Bin_Tolerance := GVL.Semi_Auto_Bin_Tolerance,
    Semi_Auto_Bin => Semi_Auto_Bin,
    semi_auto_bin_cutoff => semi_auto_bin_cutoff,
    semi_auto_bin_motor => semi_auto_bin_motor,
    Actual_Weights => Semi_Auto_Weights,
    Sequence_Complete => Semi_Auto_Complete,
    Active_Material_ID => GVL.Semi_Auto_Active_Mat,
    Active_Bin_ID => GVL.Semi_Auto_Active_Bin,
    Active_Target_Weight => Semi_Auto_Active_Target,
    Error_Code => Semi_Auto_Err,
    Status_Message => Semi_Auto_Msg
);

(* Runtime Error Mapping & Aggregation *)
IF Auto_Err <> 0 THEN
    GVL.Error_Code := Auto_Err;
    Status_Message := CONCAT('Auto Error: ', Auto_Msg);
    (* Wherever it stops, completion outputs must register TRUE *)
    Auto_Complete := TRUE;
    Semi_Auto_Complete := TRUE;
    All_Cycles_Complete := TRUE;
    GVL.Run := FALSE;
ELSIF Semi_Auto_Err <> 0 THEN
    GVL.Error_Code := Semi_Auto_Err;
    Status_Message := CONCAT('Semi-Auto Error: ', Semi_Auto_Msg);
    (* Wherever it stops, completion outputs must register TRUE *)
    Auto_Complete := TRUE;
    Semi_Auto_Complete := TRUE;
    All_Cycles_Complete := TRUE;
    GVL.Run := FALSE;
ELSIF Cycle_Manager_State = 0 THEN
    GVL.Error_Code := 0;
END_IF;

END_PROGRAM

// PLC_AC500_V3/Application/Auto_Batching_V13
FUNCTION_BLOCK Auto_Batching_V13
VAR_INPUT
    Start_Button : BOOL;      // Signal to start/resume the batching sequence
    E_Stop_Active : BOOL;     // Emergency Stop (Pause/Hold signal)
    Reset : BOOL;             // Hard reset sequence trigger
    Auto_Bin_Material_Mapping : ARRAY[1..6] OF INT; // Material index mapping for 6 bins
    Auto_Bin_Cutoff_Weights : ARRAY[1..6] OF REAL; // Cutoff weight thresholds (kg)
    Auto_Bin_Tolerance : ARRAY[1..6] OF REAL; // Tolerance weight offset values (kg)
    Inter_Bin_Delay : TIME;   // Global inter-bin delay time
    Excess_Allowed : BOOL;    // Global toggle: TRUE = skip excess check, FALSE = trigger alarm & hold
END_VAR
VAR_IN_OUT
    load_cell_value : REAL;   // Weight value read/written from load cell
END_VAR
VAR_OUTPUT
    Auto_Bin : ARRAY[1..6] OF BOOL; // Coarse feed valve outputs
    auto_bin_cutoff : ARRAY[1..6] OF BOOL; // Fine feed cutoff trigger indicators
    auto_bin_motor : ARRAY[1..6] OF BOOL; // Main conveyor motor outputs
    Actual_Weights : ARRAY[1..6] OF REAL; // Actual weight poured per silo
    Sequence_Complete : BOOL;  // Batch complete flag
    Active_Material_ID : INT;  // Currently active ingredient ID
    Active_Bin_ID : INT;       // Currently active physical Bin ID (1..6)
    Active_Target_Weight : REAL; // Recipe target weight of active bin
    Active_Live_Weight : REAL; // Live tared weight poured from active bin
    Excess_Alarm : BOOL;       // Excess weight alarm output
    Error_Code : INT;          // Active error code
    Status_Message : STRING;   // Diagnostic text message
END_VAR
VAR
    Step : INT;                // State machine index (0: Idle, 1..6: Pour, 7: Settling, 8: Complete)
    bin_last_weight : REAL;   // Baseline weight snapshot before starting current bin
    actual_bin : REAL;        // Current weight added from active bin
    target_weight : REAL;     // Target recipe weight
    cutoff_trigger_weight : REAL; // Calculated cutoff trigger threshold (Target - Cutoff)
    min_tol_weight : REAL;    // Minimum allowable tolerance (Target - Tol)
    max_tol_weight : REAL;    // Maximum allowable tolerance (Target + Tol)
    Paused_By_EStop : BOOL;    // Pause status latch
    Effective_Delay : TIME;   // Resolved delay time (defaults to T#2S if T#0S configured)
    
    Mat_Idx : INT;
    i : INT;                  // General loop index
    
    (* TIMERS FOR TRANSITIONS & DELAYS *)
    Transition_Timer : TON;
    Completion_Timer : TON;
    
    (* SELF-CONTAINED SIMULATION VARIABLES *)
    Simulation_Mode : BOOL;    // Simulation disabled for physical PLC use
    Sim_Rate : REAL;
    Sim_Timer : TON;
    Start_Sim_Weight : REAL;
    Discharge_Active : BOOL;
END_VAR

(* Auto Batching FB V13 with Real-Time Instant Excess Verification & Clean Multi-Cycle Reset *)

Effective_Delay := Inter_Bin_Delay;
IF Effective_Delay = T#0S THEN
    Effective_Delay := T#2S;
END_IF;

(* 1. HARD RESET INTERLOCK *)
IF Reset THEN
    FOR i := 1 TO 6 DO
        Auto_Bin[i] := FALSE;
        auto_bin_cutoff[i] := FALSE;
        auto_bin_motor[i] := FALSE;
        Actual_Weights[i] := 0.0;
    END_FOR;
    Sequence_Complete := FALSE;
    Active_Material_ID := 0;
    Active_Bin_ID := 0;
    Active_Target_Weight := 0.0;
    Active_Live_Weight := 0.0;
    Excess_Alarm := FALSE;
    Error_Code := 0;
    Status_Message := '';
    Paused_By_EStop := FALSE;
    Step := 0;
    
    bin_last_weight := 0.0;
    Start_Sim_Weight := 0.0;
    
    Transition_Timer(IN := FALSE);
    Completion_Timer(IN := FALSE);
    Sim_Timer(IN := FALSE);
    RETURN;
END_IF;

(* 2. E-STOP PAUSE / HOLD LOGIC *)
IF E_Stop_Active THEN
    Paused_By_EStop := TRUE;
END_IF;

IF Paused_By_EStop THEN
    FOR i := 1 TO 6 DO
        Auto_Bin[i] := FALSE;
        auto_bin_cutoff[i] := FALSE;
        auto_bin_motor[i] := FALSE;
    END_FOR;
    
    IF E_Stop_Active THEN
        Status_Message := 'Auto Paused: Emergency Stop Active!';
    ELSE
        Status_Message := 'Auto Paused: Press Start to Resume';
        IF Start_Button THEN
            Paused_By_EStop := FALSE;
        END_IF;
    END_IF;
    
    Sim_Timer(IN := FALSE);
    Transition_Timer(IN := FALSE);
    Completion_Timer(IN := FALSE);
    RETURN;
END_IF;

(* 3. SIMULATION WEIGHT MANAGEMENT (WHEN ENABLED) *)
IF Simulation_Mode THEN
    IF Step = 0 AND NOT Start_Button AND NOT Sequence_Complete THEN
        load_cell_value := 0.0;
        bin_last_weight := 0.0;
        Start_Sim_Weight := 0.0;
        Sim_Timer(IN := FALSE);
    END_IF;
    
    Discharge_Active := FALSE;
    IF Step >= 1 AND Step <= 6 THEN
        Discharge_Active := auto_bin_motor[Step];
    END_IF;
    
    IF Discharge_Active THEN
        Sim_Timer(IN := TRUE, PT := T#1000S);
        load_cell_value := Start_Sim_Weight + (TIME_TO_REAL(Sim_Timer.ET) / 1000.0) * Sim_Rate;
    ELSE
        Sim_Timer(IN := FALSE);
        Start_Sim_Weight := load_cell_value;
    END_IF;
END_IF;

(* 4. RECIPE SEQUENCE START & CYCLIC RESET *)
IF Step = 0 AND Start_Button THEN
    Step := 1;
    bin_last_weight := load_cell_value; (* Snapshot relative tare at whatever weight scale is *)
    Sequence_Complete := FALSE;
    Excess_Alarm := FALSE;
    Error_Code := 0;
    Status_Message := 'Auto Pour Started';
    Active_Target_Weight := 0.0;
    Active_Live_Weight := 0.0;
    FOR i := 1 TO 6 DO
        Actual_Weights[i] := 0.0;
        Auto_Bin[i] := FALSE;
        auto_bin_cutoff[i] := FALSE;
        auto_bin_motor[i] := FALSE;
    END_FOR;
END_IF;

(* 5. SEQUENCE CONTROL STATE MACHINE *)
CASE Step OF
    0:
        Active_Material_ID := 0;
        Active_Bin_ID := 0;
        Active_Target_Weight := 0.0;
        Active_Live_Weight := 0.0;
        Excess_Alarm := FALSE;
        Sequence_Complete := FALSE;
        FOR i := 1 TO 6 DO
            Auto_Bin[i] := FALSE;
            auto_bin_cutoff[i] := FALSE;
            auto_bin_motor[i] := FALSE;
        END_FOR;
        IF Error_Code = 0 THEN Status_Message := 'Auto Idle'; END_IF;
        
    1..6: (* DISCHARGE SILOS 1 TO 6 *)
        Mat_Idx := Auto_Bin_Material_Mapping[Step];
        
        (* Skip this step instantly if material mapping is 0 OR target weight is 0.0 kg *)
        IF Mat_Idx = 0 OR (Mat_Idx <= 20 AND GVL.Recipe_Weights[Mat_Idx] = 0.0) THEN
            IF Step = 6 THEN
                Step := 7; (* Transition directly to final settling delay *)
            ELSE
                Step := Step + 1;
            END_IF;
        ELSE
            target_weight := GVL.Recipe_Weights[Mat_Idx];
            cutoff_trigger_weight := target_weight - Auto_Bin_Cutoff_Weights[Step];
            min_tol_weight := target_weight - Auto_Bin_Tolerance[Step];
            max_tol_weight := target_weight + Auto_Bin_Tolerance[Step];
            
            Active_Target_Weight := target_weight;
            actual_bin := load_cell_value - bin_last_weight;
            Actual_Weights[Step] := actual_bin;
            Active_Live_Weight := actual_bin; (* Live tared weight of active bin *)
            
            Active_Material_ID := Mat_Idx;
            Active_Bin_ID := Step;
            
            (* Scale Overload Protection *)
            IF load_cell_value > 500.0 THEN
                Error_Code := 21;
                Status_Message := 'Error 21: Scale Overloaded!';
                Sequence_Complete := TRUE;
                Paused_By_EStop := TRUE;
            END_IF;
            
            (* Real-Time Feed & Instant Excess Alarm *)
            IF actual_bin < cutoff_trigger_weight THEN
                (* Coarse Feed *)
                Auto_Bin[Step] := TRUE;
                auto_bin_cutoff[Step] := FALSE;
                auto_bin_motor[Step] := TRUE;
                Excess_Alarm := FALSE;
                Status_Message := 'Auto Pouring (Coarse Feed)';
                
            ELSIF actual_bin < min_tol_weight THEN
                (* Fine Feed *)
                Auto_Bin[Step] := FALSE;
                auto_bin_cutoff[Step] := TRUE;
                auto_bin_motor[Step] := TRUE;
                Excess_Alarm := FALSE;
                Status_Message := 'Auto Pouring (Fine Feed)';
                
            ELSIF actual_bin > max_tol_weight THEN
                (* Excess Weight -> Instant Alarm, No Delay! *)
                Auto_Bin[Step] := FALSE;
                auto_bin_cutoff[Step] := FALSE;
                auto_bin_motor[Step] := FALSE;
                
                IF Excess_Allowed THEN
                    Excess_Alarm := FALSE;
                    Status_Message := 'Excess Weight Allowed: Advancing';
                    bin_last_weight := load_cell_value;
                    Active_Target_Weight := 0.0;
                    Active_Live_Weight := 0.0;
                    IF Step = 6 THEN
                        Step := 7;
                    ELSE
                        Step := Step + 1;
                    END_IF;
                ELSE
                    Excess_Alarm := TRUE; (* Immediate Trigger! *)
                    Status_Message := 'Excess Alarm: Weight above max tolerance! Reduce weight.';
                END_IF;
                
            ELSE
                (* In Tolerance Window [Min_Tol .. Max_Tol] *)
                Auto_Bin[Step] := FALSE;
                auto_bin_cutoff[Step] := FALSE;
                auto_bin_motor[Step] := FALSE;
                Excess_Alarm := FALSE;
                bin_last_weight := load_cell_value;
                Active_Target_Weight := 0.0;
                Active_Live_Weight := 0.0;
                
                IF Step = 6 THEN
                    Step := 7;
                ELSE
                    Step := Step + 1;
                END_IF;
            END_IF;
        END_IF;

    7: (* POST-SEQUENCE FINAL SETTLING DELAY *)
        Active_Material_ID := 0;
        Active_Bin_ID := 0;
        Active_Target_Weight := 0.0;
        Active_Live_Weight := 0.0;
        Excess_Alarm := FALSE;
        Status_Message := 'Final Settling Delay';
        Completion_Timer(IN := TRUE, PT := Effective_Delay);
        IF Completion_Timer.Q THEN
            Completion_Timer(IN := FALSE);
            Step := 8;
        END_IF;
        
    8: (* COMPLETE *)
        Active_Material_ID := 0;
        Active_Bin_ID := 0;
        Active_Target_Weight := 0.0;
        Active_Live_Weight := 0.0;
        Excess_Alarm := FALSE;
        Status_Message := 'Sequence Completed';
        Sequence_Complete := TRUE;
        
        IF NOT Start_Button THEN
            Step := 0;
            Sequence_Complete := FALSE;
            FOR i := 1 TO 6 DO
                Actual_Weights[i] := 0.0;
            END_FOR;
        END_IF;
END_CASE;

END_FUNCTION_BLOCK

// PLC_AC500_V3/Application/Semi_Auto_Batching_V13
FUNCTION_BLOCK Semi_Auto_Batching_V13
VAR_INPUT
    Start_Button : BOOL;      // Signal to start/resume the batching sequence
    E_Stop_Active : BOOL;     // Emergency Stop (Pause/Hold signal)
    Reset : BOOL;             // Hard reset sequence trigger
    Semi_Auto_Bin_Material_Mapping : ARRAY[1..10] OF INT; // Material index mapping for 10 manual silos
    Semi_Auto_Bin_Cutoff_Weights : ARRAY[1..10] OF REAL; // Cutoff weight thresholds (kg)
    Semi_Auto_Bin_Tolerance : ARRAY[1..10] OF REAL; // Tolerance weight offset values (kg)
    Inter_Bin_Delay : TIME;   // Global inter-bin delay time
    Excess_Allowed : BOOL;    // Global toggle: TRUE = skip excess check, FALSE = trigger alarm & hold
END_VAR
VAR_IN_OUT
    load_cell_value : REAL;   // Weight value read/written from load cell
END_VAR
VAR_OUTPUT
    Semi_Auto_Bin : ARRAY[1..10] OF BOOL; // Prompts/indicators for Bins 1..10
    semi_auto_bin_cutoff : ARRAY[1..10] OF BOOL; // Manual pre-cutoff indicators
    semi_auto_bin_motor : ARRAY[1..10] OF BOOL; // Main manual feeder motor outputs
    Actual_Weights : ARRAY[1..10] OF REAL; // Actual weight poured per silo
    Sequence_Complete : BOOL;  // Batch complete flag
    Active_Material_ID : INT;  // Currently active ingredient ID
    Active_Bin_ID : INT;       // Currently active physical Bin ID (1..10)
    Active_Target_Weight : REAL; // Recipe target weight of active bin
    Active_Live_Weight : REAL; // Live tared weight poured from active bin
    Excess_Alarm : BOOL;       // Excess weight alarm output
    Error_Code : INT;          // Active error code
    Status_Message : STRING;   // Diagnostic text message
END_VAR
VAR
    Step : INT;                // State machine index (0: Idle, 1..10: Pour, 31: Settling, 32: Complete)
    bin_last_weight : REAL;   // Baseline weight snapshot before starting current bin
    actual_bin : REAL;        // Current weight added from active bin
    target_weight : REAL;     // Target recipe weight
    cutoff_trigger_weight : REAL; // Calculated target threshold weight (Target - Cutoff)
    min_tol_weight : REAL;    // Minimum allowable tolerance (Target - Tol)
    max_tol_weight : REAL;    // Maximum allowable tolerance (Target + Tol)
    Paused_By_EStop : BOOL;    // Pause status latch
    Effective_Delay : TIME;   // Resolved delay time (defaults to T#2S if T#0S configured)
    
    Mat_Idx : INT;
    i : INT;                  // General loop index
    
    (* TIMERS FOR TRANSITIONS & DELAYS *)
    Transition_Timer : TON;
    Completion_Timer : TON;
    
    (* SELF-CONTAINED SIMULATION VARIABLES *)
    Simulation_Mode : BOOL;    // Simulation disabled for physical PLC use
    Sim_Rate : REAL;
    Sim_Timer : TON;
    Start_Sim_Weight : REAL;
    Discharge_Active : BOOL;
END_VAR

(* Semi-Auto Batching FB V13 with Real-Time Instant Excess Verification & Clean Multi-Cycle Reset *)

Effective_Delay := Inter_Bin_Delay;
IF Effective_Delay = T#0S THEN
    Effective_Delay := T#2S;
END_IF;

(* 1. HARD RESET INTERLOCK *)
IF Reset THEN
    FOR i := 1 TO 10 DO
        Semi_Auto_Bin[i] := FALSE;
        semi_auto_bin_cutoff[i] := FALSE;
        semi_auto_bin_motor[i] := FALSE;
        Actual_Weights[i] := 0.0;
    END_FOR;
    Sequence_Complete := FALSE;
    Active_Material_ID := 0;
    Active_Bin_ID := 0;
    Active_Target_Weight := 0.0;
    Active_Live_Weight := 0.0;
    Excess_Alarm := FALSE;
    Error_Code := 0;
    Status_Message := '';
    Paused_By_EStop := FALSE;
    Step := 0;
    
    bin_last_weight := 0.0;
    Start_Sim_Weight := 0.0;
    
    Transition_Timer(IN := FALSE);
    Completion_Timer(IN := FALSE);
    Sim_Timer(IN := FALSE);
    RETURN;
END_IF;

(* 2. E-STOP PAUSE / HOLD LOGIC *)
IF E_Stop_Active THEN
    Paused_By_EStop := TRUE;
END_IF;

IF Paused_By_EStop THEN
    FOR i := 1 TO 10 DO
        Semi_Auto_Bin[i] := FALSE;
        semi_auto_bin_cutoff[i] := FALSE;
        semi_auto_bin_motor[i] := FALSE;
    END_FOR;
    
    IF E_Stop_Active THEN
        Status_Message := 'Semi-Auto Paused: Emergency Stop Active!';
    ELSE
        Status_Message := 'Semi-Auto Paused: Press Start to Resume';
        IF Start_Button THEN
            Paused_By_EStop := FALSE;
        END_IF;
    END_IF;
    
    Sim_Timer(IN := FALSE);
    Transition_Timer(IN := FALSE);
    Completion_Timer(IN := FALSE);
    RETURN;
END_IF;

(* 3. SIMULATION WEIGHT MANAGEMENT (WHEN ENABLED) *)
IF Simulation_Mode THEN
    IF Step = 0 AND NOT Start_Button AND NOT Sequence_Complete THEN
        load_cell_value := 0.0;
        bin_last_weight := 0.0;
        Start_Sim_Weight := 0.0;
        Sim_Timer(IN := FALSE);
    END_IF;
    
    Discharge_Active := FALSE;
    IF Step >= 1 AND Step <= 10 THEN
        Discharge_Active := semi_auto_bin_motor[Step];
    END_IF;
    
    IF Discharge_Active THEN
        Sim_Timer(IN := TRUE, PT := T#1000S);
        load_cell_value := Start_Sim_Weight + (TIME_TO_REAL(Sim_Timer.ET) / 1000.0) * Sim_Rate;
    ELSE
        Sim_Timer(IN := FALSE);
        Start_Sim_Weight := load_cell_value;
    END_IF;
END_IF;

(* 4. RECIPE SEQUENCE START & CYCLIC RESET *)
IF Step = 0 AND Start_Button THEN
    Step := 1;
    bin_last_weight := load_cell_value; (* Snapshot relative tare at whatever weight scale is *)
    Sequence_Complete := FALSE;
    Excess_Alarm := FALSE;
    Error_Code := 0;
    Status_Message := 'Semi-Auto Pour Started';
    Active_Target_Weight := 0.0;
    Active_Live_Weight := 0.0;
    FOR i := 1 TO 10 DO
        Actual_Weights[i] := 0.0;
        Semi_Auto_Bin[i] := FALSE;
        semi_auto_bin_cutoff[i] := FALSE;
        semi_auto_bin_motor[i] := FALSE;
    END_FOR;
END_IF;

(* 5. SEQUENCE CONTROL STATE MACHINE *)
CASE Step OF
    0:
        Active_Material_ID := 0;
        Active_Bin_ID := 0;
        Active_Target_Weight := 0.0;
        Active_Live_Weight := 0.0;
        Excess_Alarm := FALSE;
        Sequence_Complete := FALSE;
        FOR i := 1 TO 10 DO
            Semi_Auto_Bin[i] := FALSE;
            semi_auto_bin_cutoff[i] := FALSE;
            semi_auto_bin_motor[i] := FALSE;
        END_FOR;
        IF Error_Code = 0 THEN Status_Message := 'Semi-Auto Idle'; END_IF;
        
    1..10: (* DISCHARGE SILOS 1 TO 10 *)
        Mat_Idx := Semi_Auto_Bin_Material_Mapping[Step];
        
        (* Skip this step instantly if material mapping is 0 OR target weight is 0.0 kg *)
        IF Mat_Idx = 0 OR (Mat_Idx <= 20 AND GVL.Recipe_Weights[Mat_Idx] = 0.0) THEN
            IF Step = 10 THEN
                Step := 31; (* Transition directly to final settling delay *)
            ELSE
                Step := Step + 1;
            END_IF;
        ELSE
            target_weight := GVL.Recipe_Weights[Mat_Idx];
            cutoff_trigger_weight := target_weight - Semi_Auto_Bin_Cutoff_Weights[Step];
            min_tol_weight := target_weight - Semi_Auto_Bin_Tolerance[Step];
            max_tol_weight := target_weight + Semi_Auto_Bin_Tolerance[Step];
            
            Active_Target_Weight := target_weight;
            actual_bin := load_cell_value - bin_last_weight;
            Actual_Weights[Step] := actual_bin;
            Active_Live_Weight := actual_bin; (* Live tared weight of active bin *)
            
            Active_Material_ID := Mat_Idx;
            Active_Bin_ID := Step; (* Direct 1..10 *)
            
            (* Scale Overload Protection *)
            IF load_cell_value > 500.0 THEN
                Error_Code := 21;
                Status_Message := 'Error 21: Scale Overloaded!';
                Sequence_Complete := TRUE;
                Paused_By_EStop := TRUE;
            END_IF;
            
            (* Real-Time Feed & Instant Excess Alarm *)
            IF actual_bin < cutoff_trigger_weight THEN
                (* Coarse Feed *)
                Semi_Auto_Bin[Step] := TRUE;
                semi_auto_bin_cutoff[Step] := FALSE;
                semi_auto_bin_motor[Step] := TRUE;
                Excess_Alarm := FALSE;
                Status_Message := 'Semi-Auto Pouring (Coarse Feed)';
                
            ELSIF actual_bin < min_tol_weight THEN
                (* Fine Feed *)
                Semi_Auto_Bin[Step] := FALSE;
                semi_auto_bin_cutoff[Step] := TRUE;
                semi_auto_bin_motor[Step] := TRUE;
                Excess_Alarm := FALSE;
                Status_Message := 'Semi-Auto Pouring (Fine Feed)';
                
            ELSIF actual_bin > max_tol_weight THEN
                (* Excess Weight -> Instant Alarm, No Delay! *)
                Semi_Auto_Bin[Step] := FALSE;
                semi_auto_bin_cutoff[Step] := FALSE;
                semi_auto_bin_motor[Step] := FALSE;
                
                IF Excess_Allowed THEN
                    Excess_Alarm := FALSE;
                    Status_Message := 'Excess Weight Allowed: Advancing';
                    bin_last_weight := load_cell_value;
                    Active_Target_Weight := 0.0;
                    Active_Live_Weight := 0.0;
                    IF Step = 10 THEN
                        Step := 31;
                    ELSE
                        Step := Step + 1;
                    END_IF;
                ELSE
                    Excess_Alarm := TRUE; (* Immediate Trigger! *)
                    Status_Message := 'Excess Alarm: Weight above max tolerance! Reduce weight.';
                END_IF;
                
            ELSE
                (* In Tolerance Window [Min_Tol .. Max_Tol] *)
                Semi_Auto_Bin[Step] := FALSE;
                semi_auto_bin_cutoff[Step] := FALSE;
                semi_auto_bin_motor[Step] := FALSE;
                Excess_Alarm := FALSE;
                bin_last_weight := load_cell_value;
                Active_Target_Weight := 0.0;
                Active_Live_Weight := 0.0;
                
                IF Step = 10 THEN
                    Step := 31;
                ELSE
                    Step := Step + 1;
                END_IF;
            END_IF;
        END_IF;

    31: (* POST-SEQUENCE FINAL SETTLING DELAY *)
        Active_Material_ID := 0;
        Active_Bin_ID := 0;
        Active_Target_Weight := 0.0;
        Active_Live_Weight := 0.0;
        Excess_Alarm := FALSE;
        Status_Message := 'Final Settling Delay';
        Completion_Timer(IN := TRUE, PT := Effective_Delay);
        IF Completion_Timer.Q THEN
            Completion_Timer(IN := FALSE);
            Step := 32;
        END_IF;
        
    32: (* COMPLETE *)
        Active_Material_ID := 0;
        Active_Bin_ID := 0;
        Active_Target_Weight := 0.0;
        Active_Live_Weight := 0.0;
        Excess_Alarm := FALSE;
        Status_Message := 'Sequence Completed';
        Sequence_Complete := TRUE;
        
        IF NOT Start_Button THEN
            Step := 0;
            Sequence_Complete := FALSE;
            FOR i := 1 TO 10 DO
                Actual_Weights[i] := 0.0;
            END_FOR;
        END_IF;
END_CASE;

END_FUNCTION_BLOCK

// PLC_AC500_V3/Application/batching13
PROGRAM batching13
VAR
    Auto_Ctrl : Auto_Batching_V13;
    Semi_Auto_Ctrl : Semi_Auto_Batching_V13;
    
    (* Sub-Block Diagnostic Indicators *)
    Auto_Err : INT;
    Auto_Msg : STRING;
    
    Semi_Auto_Err : INT;
    Semi_Auto_Msg : STRING;
    
    Auto_Complete : BOOL;
    Semi_Auto_Complete : BOOL;
    
    (* Repetitive Cycle Status *)
    Completed_Batch_Cycles : INT;      // Total completed batch cycle loops
    All_Cycles_Complete : BOOL;         // Indicator for full set completion
    
    (* Diagnostics & Interlocks *)
    Status_Message : STRING;
    
    i : INT;
    j : INT;
    Duplicate_Found : BOOL;
    Invalid_Material_Range : BOOL;
    Weight_Limit_Error : BOOL;
    
    (* Cycle Manager state variables *)
    Cycle_Manager_State : INT;         // State index for loop management
    Internal_FB_Start : BOOL;          // Controlled command to restart sub-blocks
END_VAR

(* 1. STARTUP CONFIGURATION, RECIPE TOTALS, AND WEIGHT CHECKS *)
Duplicate_Found := FALSE;
Invalid_Material_Range := FALSE;
Weight_Limit_Error := FALSE;

(* Calculate Auto Total Target Weight & Material Count *)
GVL.Auto_Total_Target_Weight := 0.0;
GVL.Auto_Material_Count := 0;
FOR i := 1 TO 6 DO
    (* Check 2: Out of Range (Auto) *)
    IF GVL.Auto_Bin_Material_Mapping[i] < 0 OR GVL.Auto_Bin_Material_Mapping[i] > 20 THEN
        Invalid_Material_Range := TRUE;
    END_IF;
    
    (* Check 1: Duplicate Cross-Array Material ID *)
    IF GVL.Auto_Bin_Material_Mapping[i] <> 0 AND GVL.Auto_Bin_Material_Mapping[i] <= 20 THEN
        FOR j := 1 TO 10 DO
            IF GVL.Auto_Bin_Material_Mapping[i] = GVL.Semi_Auto_Bin_Material_Mapping[j] THEN
                Duplicate_Found := TRUE;
            END_IF;
        END_FOR;
    END_IF;
    
    (* Accumulate Auto Total Target Weight and Active Count *)
    IF GVL.Auto_Bin_Material_Mapping[i] > 0 AND GVL.Auto_Bin_Material_Mapping[i] <= 20 THEN
        IF GVL.Recipe_Weights[GVL.Auto_Bin_Material_Mapping[i]] > 0.0 THEN
            GVL.Auto_Total_Target_Weight := GVL.Auto_Total_Target_Weight + GVL.Recipe_Weights[GVL.Auto_Bin_Material_Mapping[i]];
            GVL.Auto_Material_Count := GVL.Auto_Material_Count + 1;
            
            (* Check 3: Recipe weight is less than Cutoff + Tolerance *)
            IF GVL.Recipe_Weights[GVL.Auto_Bin_Material_Mapping[i]] < (GVL.Auto_Bin_Cutoff_Weights[i] + GVL.Auto_Bin_Tolerance[i]) THEN
                Weight_Limit_Error := TRUE;
            END_IF;
        END_IF;
    END_IF;
END_FOR;

(* Calculate Semi-Auto Total Target Weight & Material Count *)
GVL.Semi_Auto_Total_Target_Weight := 0.0;
GVL.Semi_Auto_Material_Count := 0;
FOR j := 1 TO 10 DO
    (* Check 2: Out of Range (Semi-Auto) *)
    IF GVL.Semi_Auto_Bin_Material_Mapping[j] < 0 OR GVL.Semi_Auto_Bin_Material_Mapping[j] > 20 THEN
        Invalid_Material_Range := TRUE;
    END_IF;
    
    (* Accumulate Semi-Auto Total Target Weight and Active Count *)
    IF GVL.Semi_Auto_Bin_Material_Mapping[j] > 0 AND GVL.Semi_Auto_Bin_Material_Mapping[j] <= 20 THEN
        IF GVL.Recipe_Weights[GVL.Semi_Auto_Bin_Material_Mapping[j]] > 0.0 THEN
            GVL.Semi_Auto_Total_Target_Weight := GVL.Semi_Auto_Total_Target_Weight + GVL.Recipe_Weights[GVL.Semi_Auto_Bin_Material_Mapping[j]];
            GVL.Semi_Auto_Material_Count := GVL.Semi_Auto_Material_Count + 1;
            
            (* Check 3: Recipe weight check (Semi-Auto) *)
            IF GVL.Recipe_Weights[GVL.Semi_Auto_Bin_Material_Mapping[j]] < (GVL.Semi_Auto_Bin_Cutoff_Weights[j] + GVL.Semi_Auto_Bin_Tolerance[j]) THEN
                Weight_Limit_Error := TRUE;
            END_IF;
        END_IF;
    END_IF;
END_FOR;

(* Configuration Error Resolution *)
IF Duplicate_Found THEN
    GVL.Error_Code := 1;
    Status_Message := 'Error 1: Duplicate Material ID mapped in Auto and Semi-Auto!';
ELSIF Invalid_Material_Range THEN
    GVL.Error_Code := 2;
    Status_Message := 'Error 2: Material Index configuration out of range (1..20)!';
ELSIF Weight_Limit_Error THEN
    GVL.Error_Code := 3;
    Status_Message := 'Error 3: Recipe weight is less than Cutoff + Tolerance!';
ELSE
    IF GVL.Error_Code <= 3 THEN
        GVL.Error_Code := 0;
    END_IF;
END_IF;

(* Abort / Hard Reset Interlock *)
IF (GVL.Error_Code >= 1 AND GVL.Error_Code <= 3) OR GVL.Reset THEN
    FOR i := 1 TO 6 DO 
        GVL.Auto_Bin[i] := FALSE; 
        GVL.auto_bin_cutoff[i] := FALSE; 
        GVL.auto_bin_motor[i] := FALSE; 
        GVL.Auto_Weights[i] := 0.0;
    END_FOR;
    
    FOR i := 1 TO 10 DO 
        GVL.Semi_Auto_Bin[i] := FALSE; 
        GVL.semi_auto_bin_cutoff[i] := FALSE; 
        GVL.semi_auto_bin_motor[i] := FALSE; 
        GVL.Semi_Auto_Weights[i] := 0.0;
    END_FOR;
    
    Internal_FB_Start := FALSE;
    Auto_Ctrl(Start_Button := FALSE, E_Stop_Active := FALSE, Reset := GVL.Reset, load_cell_value := GVL.load_cell_auto, Inter_Bin_Delay := GVL.Auto_Inter_Bin_Delay, Excess_Allowed := GVL.Auto_Excess_Allowed);
    Semi_Auto_Ctrl(Start_Button := FALSE, E_Stop_Active := FALSE, Reset := GVL.Reset, load_cell_value := GVL.load_cell_semi_auto, Inter_Bin_Delay := GVL.Semi_Auto_Inter_Bin_Delay, Excess_Allowed := GVL.Semi_Auto_Excess_Allowed);
    
    GVL.Auto_Active_Target_Weight := 0.0;
    GVL.Auto_Active_Live_Weight := 0.0;
    GVL.Semi_Auto_Active_Target_Weight := 0.0;
    GVL.Semi_Auto_Active_Live_Weight := 0.0;
    
    Auto_Complete := TRUE;
    Semi_Auto_Complete := TRUE;
    All_Cycles_Complete := TRUE;
    
    GVL.Cycle_Hold_Active := FALSE;
    GVL.Run := FALSE;
    Cycle_Manager_State := 0;
    
    IF GVL.Reset THEN
        GVL.Error_Code := 0;
        GVL.Current_Batch_Cycle := 0;
        GVL.Target_Batch_Cycles := 0;
        GVL.Start_Button := FALSE;
        Completed_Batch_Cycles := 0;
        Status_Message := 'System Reset Activated';
        Auto_Complete := FALSE;
        Semi_Auto_Complete := FALSE;
        All_Cycles_Complete := FALSE;
        
        GVL.Auto_Active_Mat := 0;
        GVL.Auto_Active_Bin := 0;
        GVL.Semi_Auto_Active_Mat := 0;
        GVL.Semi_Auto_Active_Bin := 0;
        GVL.Auto_Excess_Alarm := FALSE;
        GVL.Semi_Auto_Excess_Alarm := FALSE;
        
        (* Auto-clearing trigger: set Reset back to FALSE *)
        GVL.Reset := FALSE;
    END_IF;
    RETURN;
END_IF;


(* 2. REPETITIVE CYCLE MANAGER STATE MACHINE WITH PRE-RUN INITIAL TOLERANCE CHECK *)
CASE Cycle_Manager_State OF
    0: (* IDLE STATE *)
        Internal_FB_Start := FALSE;
        All_Cycles_Complete := FALSE;
        GVL.Cycle_Hold_Active := FALSE;
        GVL.Run := FALSE;
        IF GVL.Error_Code = 0 AND Status_Message <> 'Error: Target Batch Cycles is 0!' AND Status_Message <> 'Error 4: Scale weight exceeds Initial Tolerance!' THEN 
            Status_Message := 'System Ready'; 
        END_IF;
        
        IF GVL.Start_Button THEN
            (* Guard 1: Target_Batch_Cycles must be > 0 *)
            IF GVL.Target_Batch_Cycles <= 0 THEN
                GVL.Run := FALSE;
                Status_Message := 'Error: Target Batch Cycles is 0!';
            (* Guard 2: Check Initial Tolerance ONLY before setting Run = TRUE *)
            ELSIF (GVL.load_cell_auto > GVL.Auto_Initial_Tolerance OR GVL.load_cell_auto < (-GVL.Auto_Initial_Tolerance)) OR 
                  (GVL.load_cell_semi_auto > GVL.Semi_Auto_Initial_Tolerance OR GVL.load_cell_semi_auto < (-GVL.Semi_Auto_Initial_Tolerance)) THEN
                GVL.Run := FALSE;
                GVL.Error_Code := 4;
                Status_Message := 'Error 4: Scale weight exceeds Initial Tolerance!';
            ELSE
                GVL.Error_Code := 0;
                GVL.Current_Batch_Cycle := 1;
                Completed_Batch_Cycles := 0;
                
                Auto_Complete := FALSE;
                Semi_Auto_Complete := FALSE;
                
                GVL.Run := TRUE;
                Cycle_Manager_State := 1;
            END_IF;
        END_IF;
        
    1: (* RUN STATE (Run Sub-Blocks - Initial Tolerance is NOT checked here while pouring) *)
        Internal_FB_Start := TRUE;
        GVL.Run := TRUE;
        Status_Message := CONCAT('Running Batch Cycle ', INT_TO_STRING(GVL.Current_Batch_Cycle));
        
        (* Monitor completion of active step *)
        IF Auto_Complete AND Semi_Auto_Complete THEN
            Cycle_Manager_State := 2;
        END_IF;
        
    2: (* CHECK REPEAT CYCLE STATE *)
        Completed_Batch_Cycles := GVL.Current_Batch_Cycle;
        GVL.Run := TRUE;
        
        (* Block cycle repeat in case of active error *)
        IF GVL.Current_Batch_Cycle < GVL.Target_Batch_Cycles AND GVL.Error_Code = 0 THEN
            (* Hold cycle loop progression *)
            GVL.Cycle_Hold_Active := TRUE;
            Internal_FB_Start := FALSE; (* Reset FBs to 0 while waiting in hold *)
            Cycle_Manager_State := 5; // Go to hold wait state
        ELSE
            (* All loop cycles complete *)
            Cycle_Manager_State := 4;
        END_IF;
        
    5: (* PAUSED BETWEEN CYCLES *)
        Internal_FB_Start := FALSE; (* Keeps sub-blocks in Step 0 *)
        GVL.Run := TRUE;
        Status_Message := CONCAT('Cycle ', CONCAT(INT_TO_STRING(GVL.Current_Batch_Cycle), ' Complete. Empty scale to 0 and release Cycle Hold.'));
        
        IF NOT GVL.Cycle_Hold_Active THEN
            (* Check Initial Tolerance before starting next cycle *)
            IF (GVL.load_cell_auto > GVL.Auto_Initial_Tolerance OR GVL.load_cell_auto < (-GVL.Auto_Initial_Tolerance)) OR 
               (GVL.load_cell_semi_auto > GVL.Semi_Auto_Initial_Tolerance OR GVL.load_cell_semi_auto < (-GVL.Semi_Auto_Initial_Tolerance)) THEN
                GVL.Run := FALSE;
                GVL.Error_Code := 4;
                Status_Message := 'Error 4: Scale weight exceeds Initial Tolerance!';
                GVL.Cycle_Hold_Active := TRUE; (* Keep hold active until scale is emptied *)
            ELSE
                GVL.Error_Code := 0;
                GVL.Current_Batch_Cycle := GVL.Current_Batch_Cycle + 1;
                Auto_Complete := FALSE;
                Semi_Auto_Complete := FALSE;
                Cycle_Manager_State := 1; (* Start next cycle! *)
            END_IF;
        END_IF;
        
    4: (* SEQUENCE FULLY COMPLETED STATE *)
        Internal_FB_Start := FALSE;
        All_Cycles_Complete := TRUE;
        GVL.Run := FALSE;
        GVL.Start_Button := FALSE; (* Auto-turn off Start_Button when process completes! *)
        Status_Message := 'All Batch Cycles Completed';
        
        Cycle_Manager_State := 0;
END_CASE;


(* 3. CONCURRENT EXECUTION OF FB INSTANCES WITH GVL ARRAYS & LIVE ACTIVE WEIGHTS *)
Auto_Ctrl(
    Start_Button := Internal_FB_Start,
    E_Stop_Active := GVL.E_Stop_Active,
    Reset := GVL.Reset,
    load_cell_value := GVL.load_cell_auto,
    Auto_Bin_Material_Mapping := GVL.Auto_Bin_Material_Mapping,
    Auto_Bin_Cutoff_Weights := GVL.Auto_Bin_Cutoff_Weights,
    Auto_Bin_Tolerance := GVL.Auto_Bin_Tolerance,
    Inter_Bin_Delay := GVL.Auto_Inter_Bin_Delay,
    Excess_Allowed := GVL.Auto_Excess_Allowed,
    Auto_Bin => GVL.Auto_Bin,
    auto_bin_cutoff => GVL.auto_bin_cutoff,
    auto_bin_motor => GVL.auto_bin_motor,
    Actual_Weights => GVL.Auto_Weights,
    Sequence_Complete => Auto_Complete,
    Active_Material_ID => GVL.Auto_Active_Mat,
    Active_Bin_ID => GVL.Auto_Active_Bin,
    Active_Target_Weight => GVL.Auto_Active_Target_Weight,
    Active_Live_Weight => GVL.Auto_Active_Live_Weight,
    Excess_Alarm => GVL.Auto_Excess_Alarm,
    Error_Code => Auto_Err,
    Status_Message => Auto_Msg
);

Semi_Auto_Ctrl(
    Start_Button := Internal_FB_Start,
    E_Stop_Active := GVL.E_Stop_Active,
    Reset := GVL.Reset,
    load_cell_value := GVL.load_cell_semi_auto,
    Semi_Auto_Bin_Material_Mapping := GVL.Semi_Auto_Bin_Material_Mapping,
    Semi_Auto_Bin_Cutoff_Weights := GVL.Semi_Auto_Bin_Cutoff_Weights,
    Semi_Auto_Bin_Tolerance := GVL.Semi_Auto_Bin_Tolerance,
    Inter_Bin_Delay := GVL.Semi_Auto_Inter_Bin_Delay,
    Excess_Allowed := GVL.Semi_Auto_Excess_Allowed,
    Semi_Auto_Bin => GVL.Semi_Auto_Bin,
    semi_auto_bin_cutoff => GVL.semi_auto_bin_cutoff,
    semi_auto_bin_motor => GVL.semi_auto_bin_motor,
    Actual_Weights => GVL.Semi_Auto_Weights,
    Sequence_Complete => Semi_Auto_Complete,
    Active_Material_ID => GVL.Semi_Auto_Active_Mat,
    Active_Bin_ID => GVL.Semi_Auto_Active_Bin,
    Active_Target_Weight => GVL.Semi_Auto_Active_Target_Weight,
    Active_Live_Weight => GVL.Semi_Auto_Active_Live_Weight,
    Excess_Alarm => GVL.Semi_Auto_Excess_Alarm,
    Error_Code => Semi_Auto_Err,
    Status_Message => Semi_Auto_Msg
);

(* Runtime Error Mapping & Aggregation *)
IF Auto_Err <> 0 THEN
    GVL.Error_Code := Auto_Err;
    Status_Message := CONCAT('Auto Error: ', Auto_Msg);
    Auto_Complete := TRUE;
    Semi_Auto_Complete := TRUE;
    All_Cycles_Complete := TRUE;
    GVL.Run := FALSE;
    GVL.Start_Button := FALSE;
ELSIF Semi_Auto_Err <> 0 THEN
    GVL.Error_Code := Semi_Auto_Err;
    Status_Message := CONCAT('Semi-Auto Error: ', Semi_Auto_Msg);
    Auto_Complete := TRUE;
    Semi_Auto_Complete := TRUE;
    All_Cycles_Complete := TRUE;
    GVL.Run := FALSE;
    GVL.Start_Button := FALSE;
ELSIF Cycle_Manager_State = 0 AND GVL.Error_Code <= 3 THEN
    GVL.Error_Code := 0;
END_IF;

END_PROGRAM

(* text list Diag_IO_Bus (id | default | en | de | fr | es | zh)
  Err_1037 | Test error | Test error | Testfehler |  |  | 测试错误
  Err_12 | Test pulse error -> Check wiring and sensor | Test pulse error -> Check wiring and sensor | Testimpuls-Fehler -> Verdrahtung und Sensor prüfen |  |  | 测试脉冲错误 -> 检查接线和传感器
  Err_13 | Test pulse cross-talk error -> Check wiring and sensor. If this error persists, replace I/O module. Contact ABB technical support. | Test pulse cross-talk error -> Check wiring and sensor. If this error persists, replace I/O module. Contact ABB technical support. | Fehler Testimpuls Kanalübersprechen  -> Verdrahtung und Sensor prüfen. Falls der Fehler weiterhin besteht, E/A-Modul austauschen. Technischen Support von ABB kontaktieren. |  |  | 测试脉冲串扰错误 -> 检查接线和传感器. 如果此错误仍然存在，请更换 I/O 模块. 联系 ABB 技术支持.
  Err_16128 | Failed max wait run | Failed max wait run | Lauf max. Warten fehlgeschlagen |  |  | 最大等待运行失败
  Err_16129 | Critical error, see log | Critical error, see log | Kritischer Fehler, siehe Protokoll |  |  | 严重错误，请参阅日志
  Err_16130 | Fatal error, see log | Fatal error, see log | Schwerwiegender Fehler, siehe Protokoll |  |  | 致命错误，请参阅日志
  Err_16131 | Timeout -> Replace I/O module | Timeout -> Replace I/O module | Timeout -> E/A-Modul austauschen |  |  | 超时 -> 更换 I/O 模块
  Err_16133 | Output data size mismatch | Output data size mismatch | Diskrepanz Ausgangsdatengröße |  |  | 输出数据大小不匹配
  Err_16134 | Input data size mismatch | Input data size mismatch | Diskrepanz Eingangsdatengröße |  |  | 输入数据大小不匹配
  Err_16137 | Overflow diagnosis buffer -> Restart | Overflow diagnosis buffer -> Restart | Überlauf Diagnosepuffer -> Neu Starten |  |  | 诊断缓冲区溢出 -> 重新启动
  Err_16138 | Non-safety I/O: Voltage overflow at outputs (above UP3 level), Safety I/O: Process voltage too high -> Check terminals / Check process voltage | Non-safety I/O: Voltage overflow at outputs (above UP3 level), Safety I/O: Process voltage too high -> Check terminals / Check process voltage | Standard-E/A: Spannungsüberlauf an Ausgängen (über UP3-Niveau), Sicherheits-E/A: Prozessspannung zu hoch -> Terminals prüfen / Prozessspannung prüfen |  |  | 非安全 I/O：输出端电压溢出（高于 UP3 电平），安全 I/O：过程电压过高 -> 检查终端 / 检查过程电压
  Err_16139 | Process voltage UP or UP3 too low -> Check process voltage | Process voltage UP or UP3 too low -> Check process voltage | Prozessspannung UP oder UP3 zu niedrig -> Prozessspannung prüfen |  |  | 过程电压 UP 或 UP3 过低 -> 检查过程电压
  Err_16145 | Error setting parameters | Error setting parameters | Fehlereinstellungsparameter |  |  | 设置参数时出错
  Err_16146 | Plausibility check failed (iParameter) -> Check configuration | Plausibility check failed (iParameter) -> Check configuration | Plausibilitätsprüfung fehlgeschlagen (iParameter) -> Konfiguration überprüfen |  |  | 合理性检查失败（i 参数） -> 检查配置
  Err_16147 | Checksum error -> Non-safety I/O: Replace I/O module. Safety I/O: Check safety configuration and CRCs for I- and F-Parameters. | Checksum error -> Non-safety I/O: Replace I/O module. Safety I/O: Check safety configuration and CRCs for I- and F-Parameters. | Prüfsummenfehler -> Standard-E/A: E/A-Modul austauschen. Sicherheits-E/A: Sicherheitskonfiguration und CRCs auf I- und F-Parameter prüfen. |  |  | 检校验和错误 -> 非安全 I/O：更换 I/O 模块. 安全 I/O：检查 I 参数和 F 参数的安全配置和 CRC.
  Err_16148 | PROFIsafe communication error -> Restart I/O module. If this error persists, contact ABB technical support. | PROFIsafe communication error -> Restart I/O module. If this error persists, contact ABB technical support. | PROFIsafe-Kommunikationsfehler -> E/A-Modul neu starten. Falls der Fehler weiterhin besteht, technischen Support von ABB kontaktieren. |  |  | PROFIsafe 通信错误 -> 重新启动 I/O 模块. 如果此错误仍然存在，请联系 ABB 技术支持.
  Err_16149 | No module data | No module data | Keine Moduldaten |  |  | 无模块数据
  Err_16153 | PROFIsafe watchdog timed out -> Restart I/O module. If this error persists, increase PROFIsafe watchdog time. | PROFIsafe watchdog timed out -> Restart I/O module. If this error persists, increase PROFIsafe watchdog time. | Timeout von PROFIsafe-Watchdog -> E/A-Modul neu starten. Falls der Fehler weiterhin besteht, PROFIsafe-Watchdog-Zeit verlängern. |  |  | PROFIsafe 看门狗超时 -> 重新启动 I/O 模块. 如果此错误仍然存在，请增加 PROFIsafe 看门狗时间.
  Err_16154 | Size of parameters expected by module differs from size provided by configuration -> Check master or configuration | Size of parameters expected by module differs from size provided by configuration -> Check master or configuration | Vom Modul erwartete Parametergröße weicht von der in der Konfiguration angegebenen Größe ab -> Master oder Konfiguration überprüfen |  |  | 模块期望的参数大小与配置提供的参数大小不同 -> 检查主设备或配置
  Err_16156 | F-Parameter configuration and address switch value do not match -> Check I/O module F-Parameter configuration and module address switch value. | F-Parameter configuration and address switch value do not match -> Check I/O module F-Parameter configuration and module address switch value. | Konfiguration für F-Parameter und Wert des Adressschalters stimmen nicht überein -> Konfiguration für F-Parameter des E/A-Moduls und Wert des Adressschalters überprüfen. |  |  | F 参数配置和地址开关值不匹配 -> 检查 I/O 模块 F 参数配置和模块地址开关值.
  Err_16158 | Type of present module does not match configuration | Type of present module does not match configuration | Typ des vorhandenen Moduls stimmt nicht mit Konfiguration überein |  |  | 当前模块类型与配置不匹配
  Err_16159 | Configured number of modules differs from found ones | Configured number of modules differs from found ones | Konfigurierte Anzahl von Modulen weicht von Anzahl gefundener Module ab |  |  | 配置的模块数量与找到的模块数量不同
  Err_16160 | At least one module failed during configuration | At least one module failed during configuration | Mindestens ein Modul während Konfiguration ausgefallen |  |  | 配置期间至少有一个模块发生故障
  Err_16164 | Internal data exchange failure -> Replace I/O module | Internal data exchange failure -> Replace I/O module | Fehler interner Datenaustausch -> E/A-Modul austauschen |  |  | 内部数据交换失败 -> 更换 I/O 模块
  Err_16168 | Different hard-/firmware versions in the module -> Replace I/O module | Different hard-/firmware versions in the module -> Replace I/O module | Unterschiedliche Hardware-/Firmware-Versionen im Modul -> E/A-Modul austauschen |  |  | 模块中的硬件/固件版本不同 -> 更换 I/O 模块
  Err_16171 | Internal error -> Replace I/O module | Internal error -> Replace I/O module | Interner Fehler -> E/A-Modul austauschen |  |  | 内部错误 -> 更换 I/O 模块
  Err_16172 | Has not passed factory test | Has not passed factory test | Hat Werksprüfung nicht bestanden |  |  | 未通过出厂测试
  Err_16173 | No process voltage UP or UP3 -> Check process voltage | No process voltage UP or UP3 -> Check process voltage | Keine Prozessspannung UP oder UP3 -> Prozessspannung prüfen |  |  | 无过程电压 UP 或 UP3 -> 检查过程电压
  Err_16175 | Sensor voltage too low | Sensor voltage too low | Sensorspannung zu niedrig |  |  | 传感器电压过低
  Err_16194 | Fatal error, not running any more | Fatal error, not running any more | Schwerwiegender Fehler, Ausführung gestoppt |  |  | 致命错误，不再运行
  Err_16246 | Failed to start the parameterization of modules | Failed to start the parameterization of modules | Starten von Parametrierung für Module fehlgeschlagen |  |  | 无法启动模块的参数化
  Err_16247 | Failed setting parameters | Failed setting parameters | Einstellen von Parametern fehlgeschlagen |  |  | 设置参数失败
  Err_16248 | Failed setting expected module | Failed setting expected module | Einstellen des erwarteten Moduls fehlgeschlagen |  |  | 设置预期模块失败
  Err_16254 | Size of parameters expected by module differs from size provided by configuration | Size of parameters expected by module differs from size provided by configuration | Vom Modul erwartete Parametergröße weicht von der in der Konfiguration angegebenen Größe ab |  |  | 模块期望的参数大小与配置提供的参数大小不同
  Err_18 | Test error | Test error | Testfehler |  |  | 测试错误
  Err_25 | Stuck at error -> Check I/O module wiring. Restart I/O module, if needed. If this error persists, replace I/O module. | Stuck at error -> Check I/O module wiring. Restart I/O module, if needed. If this error persists, replace I/O module. | Hängengeblieben bei Fehler -> Verdrahtung des E/A-Moduls überprüfen. Bei Bedarf E/A-Modul neu starten. Falls der Fehler weiterhin besteht, E/A-Modul austauschen. |  |  | 卡在错误处 -> 检查 I/O 模块接线. 如果需要，重新启动 I/O 模块. 如果此错误仍然存在，请更换 I/O 模块.
  Err_257 | Wrong measurement, false temperature at the compensation channel | Wrong measurement, false temperature at the compensation channel | Falscher Messwert, falsche Temperatur an Kompensationskanal |  |  | 测量值错误，补偿通道温度错误
  Err_258 | AI531: Wrong measurement; potential difference is too high; CD522: PWM duty cycle out of duty area | AI531: Wrong measurement; potential difference is too high; CD522: PWM duty cycle out of duty area | AI531: Falscher Messwert; Potenzialdifferenz zu hoch; CD522: PWM-Einschaltdauer außerhalb des Einschaltbereichs |  |  | AI531：测量错误; 电位差过高; CD522: PWM 占空比超出占空比范围
  Err_260 | Measurement overflow -> Check channel wiring and sensor power supply | Measurement overflow -> Check channel wiring and sensor power supply | Messwertüberschreitung -> Kanalverdrahtung und Spannungsversorgung des Sensors prüfen |  |  | 测量值溢出 -> 检查通道接线和传感器电源
  Err_263 | Measurement underflow -> Check channel wiring and sensor power supply | Measurement underflow -> Check channel wiring and sensor power supply | Messwertunterschreitung -> Kanalverdrahtung und Spannungsversorgung des Sensors prüfen |  |  | 测量值下溢 -> 检查通道接线和传感器电源
  Err_266 | Short circuit and cut wire or "out of range" | Short circuit and cut wire or "out of range" | Kurzschluss und Drahtbruch oder „außerhalb des zulässigen Bereichs“ |  |  | 短路和断线或“超出范围”
  Err_267 | Output/process voltage too low | Output/process voltage too low | Ausgangs-/Prozessspannung zu gering |  |  | 输出/过程电压过低
  Err_273 | Test error | Test error | Testfehler |  |  | 测试错误
  Err_28 | Cross-talk error -> Check I/O module wiring. Restart I/O module, if needed. If this error persists, replace I/O module. | Cross-talk error -> Check I/O module wiring. Restart I/O module, if needed. If this error persists, replace I/O module. | Fehler Kanalübersprechen -> Verdrahtung des E/A-Moduls überprüfen. Bei Bedarf E/A-Modul neu starten. Falls der Fehler weiterhin besteht, E/A-Modul austauschen. |  |  | 串扰错误 -> 检查 I/O 模块接线. 如果需要，重新启动 I/O 模块. 如果此错误仍然存在，请更换 I/O 模块.
  Err_3 | Discrepancy time expired -> Check discrepancy time value, channel wiring and sensor. | Discrepancy time expired -> Check discrepancy time value, channel wiring and sensor. | Diskrepanzzeit abgelaufen -> Diskrepanzzeit-Wert, Kanalverdrahtung und Sensor überprüfen. |  |  | 偏差时间已过 -> 检查差异时间值、通道接线和传感器.
  Err_303 | Short circuit at analog input -> Check channel wiring | Short circuit at analog input -> Check channel wiring | Kurzschluss an Analogeingang -> Kanalverdrahtung prüfen |  |  | 模拟输入端短路 -> 检查通道接线
  Err_304 | Analog value overflow or broken wire at an analog input -> Check value or check terminals | Analog value overflow or broken wire at an analog input -> Check value or check terminals | Analogwert-Überlauf oder Drahtbruch an Analogeingang -> Wert oder Terminals prüfen |  |  | 模拟输入端模拟值溢出或断线 -> 检查值或检查终端
  Err_311 | Value difference too high -> Adjust tolerance window for channels. Check channel wiring and sensor configuration. | Value difference too high -> Adjust tolerance window for channels. Check channel wiring and sensor configuration. | Wertdifferenz zu groß -> Toleranzfenster für Kanäle einstellen. Kanalverdrahtung und Sensorkonfiguration prüfen. |  |  | 值差异过大 -> 调整通道的容差范围. 检查通道接线和传感器配置.
  Err_524 | Stuck at error | Stuck at error | Hängengeblieben bei Fehler |  |  | 卡在错误处
  Err_525 | Readback error -> Check I/O module wiring. Restart I/O module, if needed. If this error persists, replace I/O module. | Readback error -> Check I/O module wiring. Restart I/O module, if needed. If this error persists, replace I/O module. | Fehler Rücklesen -> Verdrahtung des E/A-Moduls überprüfen. Bei Bedarf E/A-Modul neu starten. Falls der Fehler weiterhin besteht, E/A-Modul austauschen. |  |  | 回读错误 -> 检查 I/O 模块接线. 如果需要，重新启动 I/O 模块. 如果此错误仍然存在，请更换 I/O 模块.
  Err_530 | Class 3: Cross-talk error; Class 4: Internal fuse at 0V is defect. 0V not connected with GND -> Check I/O module wiring. Restart I/O module, if needed. If this error persists, replace I/O module. | Class 3: Cross-talk error; Class 4: Internal fuse at 0V is defect. 0V not connected with GND -> Check I/O module wiring. Restart I/O module, if needed. If this error persists, replace I/O module. | Klasse 3: Fehler Kanalübersprechen; Klasse 4: Interne Sicherung an 0 V defekt. 0 V nicht an GND angeschlossen -> Verdrahtung des E/A-Moduls überprüfen. Bei Bedarf E/A-Modul neu starten. Falls der Fehler weiterhin besteht, E/A-Modul austauschen. |  |  | 3 级：串扰错误; 4 级：0V 时内部保险丝有缺陷. 0V 未连接 GND -> 检查 I/O 模块接线. 如果需要，重新启动 I/O 模块. 如果此错误仍然存在，请更换 I/O 模块.
  Err_540 | Test error | Test error | Testfehler |  |  | 测试错误
  Err_555 | Internal error | Internal error | Interner Fehler |  |  | 内部错误
  Err_559 | Short circuit at digital output -> Check channel wiring | Short circuit at digital output -> Check channel wiring | Kurzschluss an Digitalausgang -> Kanalverdrahtung prüfen |  |  | 数字输出端短路 -> 检查通道接线
  Err_772 | Measurement overflow -> Check channel wiring | Measurement overflow -> Check channel wiring | Messwertüberschreitung -> Kanalverdrahtung prüfen |  |  | 测量值溢出 -> 检查通道接线
  Err_775 | Measurement underflow at analog input -> Check channel wiring | Measurement underflow at analog input -> Check channel wiring | Messwertunterschreitung an Analogausgang -> Kanalverdrahtung prüfen |  |  | 模拟输入端测量值下溢 -> 检查通道接线
  Err_796 | Different configuration | Different configuration | Abweichende Konfiguration |  |  | 配置不同
  Err_8480 | Not supported protocol variant | Not supported protocol variant | Nicht unterstützte Protokollvariante |  |  | 不支持的协议变体
  Err_8482 | Class 2: Timeout while initializing; Class 4: Timeout while waiting for ready status | Class 2: Timeout while initializing; Class 4: Timeout while waiting for ready status | Klasse 2: Timeout bei Initialisierung; Klasse 4: Timeout beim Warten auf Status „Bereit“ |  |  | 2 级：初始化超时; 4 级：等待就绪状态超时
  Err_8483 | Timeout during parameterization | Timeout during parameterization | Timeout bei Parametrierung |  |  | 参数化期间超时
  Err_8707 | PROFIsafe watchdog timed out | PROFIsafe watchdog timed out | Timeout von PROFIsafe-Watchdog |  |  | PROFIsafe 看门狗超时
  Err_8708 | Overvoltage | Overvoltage | Überspannung |  |  | 过电压
  Err_8711 | Undervoltage | Undervoltage | Unterspannung |  |  | 欠电压
  Err_8722 | Internal error | Internal error | Interner Fehler |  |  | 内部错误
  Err_8723 | Checksum error has occured in iParameters | Checksum error has occured in iParameters | Prüfsummenfehler in iParameter |  |  | i 参数中出现校验和错误
  Err_8724 | PROFIsafe communication error | PROFIsafe communication error | PROFIsafe-Kommunikationsfehler |  |  | PROFIsafe 通信错误
  Err_8732 | Internal error | Internal error | Interner Fehler |  |  | 内部错误
  Err_8747 | Internal runtime error | Internal runtime error | Interner Laufzeitfehler |  |  | 内部运行时错误
  Err_8961 | Wrong parameter value, check configuration | Wrong parameter value, check configuration | Falscher Parameterwert, Konfiguration prüfen |  |  | 参数值错误，请检查配置
  Err_8979 | Checksum error has occured in iParameter or F-Parameters | Checksum error has occured in iParameter or F-Parameters | Prüfsummenfehler in iParameter oder F-Parametern |  |  | i 参数或 F 参数中出现校验和错误
  Err_8986 | Invalid configuration -> Check modules and parameterization | Invalid configuration -> Check modules and parameterization | Ungültige Konfiguration -> Module und Parametrierung prüfen |  |  | 配置无效 -> 检查模块和参数化
  Err_8988 | F-Parameter configuration and address switch value do not match -> Check I/O module F-Parameter configuration and module address switch value. | F-Parameter configuration and address switch value do not match -> Check I/O module F-Parameter configuration and module address switch value. | Konfiguration für F-Parameter und Wert des Adressschalters stimmen nicht überein -> Konfiguration für F-Parameter des E/A-Moduls und Wert des Adressschalters überprüfen. |  |  | F 参数配置和地址开关值不匹配 -> 检查 I/O 模块 F 参数配置和模块地址开关值.
  Err_9249 | Timeout while waiting for Reset | Timeout while waiting for Reset | Timeout beim Warten auf Zurücksetzen |  |  | 等待重置时超时
  Err_9258 | Breakdown, communication lost | Breakdown, communication lost | Ausfall, Kommunikation unterbrochen |  |  | 故障，通信中断
  Err_9480 | I/O module removed from hotswap terminal unit or defective module on hotswap terminal unit -> Plug I/O module, replace I/O module | I/O module removed from hotswap terminal unit or defective module on hotswap terminal unit -> Plug I/O module, replace I/O module | E/A-Modul von Hotswap-Terminal-Einheit entfernt oder defektes Modul an Hotswap-Terminal-Einheit -> E/A-Modul einstecken, E/A-Modul austauschen |  |  | I/O 模块已从热插拔终端单元上拔下，或热插拔终端单元上的模块有故障 -> 插入 I/O 模块，更换 I/O 模块
  Err_9500 | Wrong I/O module plugged on hotswap terminal unit -> Remove wrong I/O module and plug projected I/O module | Wrong I/O module plugged on hotswap terminal unit -> Remove wrong I/O module and plug projected I/O module | Falsches E/A-Modul an Hotwwap-Terminal-Einheit eingesteckt -> Falsches E/A-Modul entfernen oder projektiertes E/A-Modul einstecken |  |  | 热插拔终端单元上插入了错误的 I/O 模块 -> 拔出错误的 I/O 模块并插入预计的 I/O 模块
  Err_9514 | No communication with I/O module on hotswap terminal unit -> Replace I/O module | No communication with I/O module on hotswap terminal unit -> Replace I/O module | Keine Kommunikation mit E/A-Modul an Hotswap-Terminal-Einheit -> E/A-Modul austauschen |  |  | 无法与热插拔终端单元上的 I/O 模块通信 -> 更换 I/O 模块
  Err_9526 | I/O module does not support hotswap functionality -> Power off system and replace I/O module | I/O module does not support hotswap functionality -> Power off system and replace I/O module | E/A-Modul unterstützt keine Hotswap-Funktion -> System abschalten und E/A-Modul austauschen |  |  | I/O 模块不支持热插拔功能 -> 关闭系统电源并更换 I/O 模块
  Err_9736 | hotswap terminal unit required but not found | hotswap terminal unit required but not found | Hotswap-Terminal-Einheit erforderlich, jedoch nicht gefunden |  |  | 需要热插拔终端单元但未找到
  Err_9764 | Defective hotswap terminal unit | Defective hotswap terminal unit | Defekte Hotswap-Terminal-Einheit |  |  | 热插拔终端单元有缺陷
  Err_9770 | No communication with hotswap terminal unit -> Restart, if error persists replace terminal unit | No communication with hotswap terminal unit -> Restart, if error persists replace terminal unit | Keine Kommunikation mit Hotswap-Terminal-Einheit -> Neu starten, falls Fehler weiterhin besteht, Terminal-Einheit austauschen |  |  | 无法与热插拔终端单元通信 -> 重新启动，如果错误仍然存在，请更换终端单元
  Hwd_14 | I/O bus | I/O bus | E/A-Bus |  |  | I/O 总线
  Sub1_ | Module | Module | Modul |  |  | 模块
  Sub2_ | Channel | Channel | Kanal |  |  | 通道 *)

